   DATA[261,19] := 2.0;
   DATA[261,20] := 148.808;
   DATA[261,21] := 155.9087;
   DATA[261,22] := 1.718643;
   DATA[261,23] := 962.9838;
   DATA[261,24] := 2.0;
   DATA[261,25] := 2.0;
   DATA[261,26] := 7.876058;
   DATA[261,27] := 144.9885;
   DATA[261,28] := 264.0989;
   DATA[261,29] := 12.15073;
   DATA[261,30] := 1.730069;
   DATA[261,31] := 1.257846;
   DATA[261,32] := 0.7351407;
   DATA[261,33] := 0.3077859;
   DATA[261,34] := 2.0;
   DATA[261,35] := 251.0414;
   DATA[261,36] := 1.649953;
   DATA[261,37] := 189.8231;
   DATA[261,38] := 0.000128152;
   DATA[261,39] := 1.0;
   DATA[262,0] := 2.540755;
   DATA[262,1] := 527.243;
   DATA[262,2] := 2.0;
   DATA[262,3] := 2.0;
   DATA[262,4] := 262.0802;
   DATA[262,5] := 8.393873;
   DATA[262,6] := 328.2748;
   DATA[262,7] := 2.444623;
   DATA[262,8] := 2.0;
   DATA[262,9] := 2.0;
   DATA[262,10] := 2.0;
   DATA[262,11] := 19.62033;
   DATA[262,12] := 2.213496;
   DATA[262,13] := 968.2213;
   DATA[262,14] := 1.0;
   DATA[262,15] := 2.0;
   DATA[262,16] := 1.0;
   DATA[262,17] := 1.0;
   DATA[262,18] := 1.0;
   DATA[262,19] := 2.0;
   DATA[262,20] := 148.808;
   DATA[262,21] := 155.9344;
   DATA[262,22] := 1.719284;
   DATA[262,23] := 963.253;
   DATA[262,24] := 2.0;
   DATA[262,25] := 2.0;
   DATA[262,26] := 7.876058;
   DATA[262,27] := 144.9885;
   DATA[262,28] := 264.0989;
   DATA[262,29] := 12.15073;
   DATA[262,30] := 1.73071;
   DATA[262,31] := 1.254515;
   DATA[262,32] := 0.7351407;
   DATA[262,33] := 0.3077859;
   DATA[262,34] := 2.0;
   DATA[262,35] := 251.0414;
   DATA[262,36] := 1.649953;
   DATA[262,37] := 189.8231;
   DATA[262,38] := 0.000128152;
   DATA[262,39] := 1.0;
   DATA[263,0] := 2.577587;
   DATA[263,1] := 527.4393;
   DATA[263,2] := 2.0;
   DATA[263,3] := 2.0;
   DATA[263,4] := 262.0802;
   DATA[263,5] := 8.393873;
   DATA[263,6] := 328.121;
   DATA[263,7] := 2.444623;
   DATA[263,8] := 2.0;
   DATA[263,9] := 2.0;
   DATA[263,10] := 2.0;
   DATA[263,11] := 19.62033;
   DATA[263,12] := 2.214137;
   DATA[263,13] := 968.6218;
   DATA[263,14] := 1.0;
   DATA[263,15] := 2.0;
   DATA[263,16] := 1.0;
   DATA[263,17] := 1.0;
   DATA[263,18] := 1.0;
   DATA[263,19] := 2.0;
   DATA[263,20] := 148.808;
   DATA[263,21] := 155.9344;
   DATA[263,22] := 1.719284;
   DATA[263,23] := 963.4453;
   DATA[263,24] := 2.0;
   DATA[263,25] := 2.0;
   DATA[263,26] := 7.876058;
   DATA[263,27] := 144.9885;
   DATA[263,28] := 264.0989;
   DATA[263,29] := 12.15073;
   DATA[263,30] := 1.73071;
   DATA[263,31] := 1.257205;
   DATA[263,32] := 0.7351407;
   DATA[263,33] := 0.3068251;
   DATA[263,34] := 2.0;
   DATA[263,35] := 251.0414;
   DATA[263,36] := 1.649953;
   DATA[263,37] := 189.8231;
   DATA[263,38] := 0.000128152;
   DATA[263,39] := 1.0;
   DATA[264,0] := 2.6157;
   DATA[264,1] := 527.7534;
   DATA[264,2] := 2.0;
   DATA[264,3] := 2.0;
   DATA[264,4] := 262.0802;
   DATA[264,5] := 8.393873;
   DATA[264,6] := 328.121;
   DATA[264,7] := 2.44411;
   DATA[264,8] := 2.0;
   DATA[264,9] := 2.0;
   DATA[264,10] := 2.0;
   DATA[264,11] := 19.64594;
   DATA[264,12] := 2.214137;
   DATA[264,13] := 968.5818;
   DATA[264,14] := 1.0;
   DATA[264,15] := 2.0;
   DATA[264,16] := 1.0;
   DATA[264,17] := 1.0;
   DATA[264,18] := 1.0;
   DATA[264,19] := 2.0;
   DATA[264,20] := 148.808;
   DATA[264,21] := 155.9344;
   DATA[264,22] := 1.719284;
   DATA[264,23] := 963.4068;
   DATA[264,24] := 2.0;
   DATA[264,25] := 2.0;
   DATA[264,26] := 7.876058;
   DATA[264,27] := 144.9885;
   DATA[264,28] := 264.0989;
   DATA[264,29] := 12.15073;
   DATA[264,30] := 1.729557;
   DATA[264,31] := 1.261944;
   DATA[264,32] := 0.7351407;
   DATA[264,33] := 0.3068251;
   DATA[264,34] := 2.0;
   DATA[264,35] := 251.1055;
   DATA[264,36] := 1.649953;
   DATA[264,37] := 189.8231;
   DATA[264,38] := 0.000128152;
   DATA[264,39] := 1.0;
   DATA[265,0] := 2.637799;
   DATA[265,1] := 527.9496;
   DATA[265,2] := 2.0;
   DATA[265,3] := 2.0;
   DATA[265,4] := 262.0802;
   DATA[265,5] := 8.393873;
   DATA[265,6] := 328.121;
   DATA[265,7] := 2.4427;
   DATA[265,8] := 2.0;
   DATA[265,9] := 2.0;
   DATA[265,10] := 2.0;
   DATA[265,11] := 19.66835;
   DATA[265,12] := 2.214137;
   DATA[265,13] := 968.6218;
   DATA[265,14] := 1.0;
   DATA[265,15] := 2.0;
   DATA[265,16] := 1.0;
   DATA[265,17] := 1.0;
   DATA[265,18] := 1.0;
   DATA[265,19] := 2.0;
   DATA[265,20] := 148.808;
   DATA[265,21] := 155.9344;
   DATA[265,22] := 1.719284;
   DATA[265,23] := 963.1761;
   DATA[265,24] := 2.0;
   DATA[265,25] := 2.0;
   DATA[265,26] := 7.876058;
   DATA[265,27] := 144.9885;
   DATA[265,28] := 264.0989;
   DATA[265,29] := 12.15073;
   DATA[265,30] := 1.729172;
   DATA[265,31] := 1.277699;
   DATA[265,32] := 0.7351407;
   DATA[265,33] := 0.3063127;
   DATA[265,34] := 2.0;
   DATA[265,35] := 251.1055;
   DATA[265,36] := 1.649953;
   DATA[265,37] := 189.8071;
   DATA[265,38] := 0.000128152;
   DATA[265,39] := 1.0;
   DATA[266,0] := 2.656055;
   DATA[266,1] := 527.7534;
   DATA[266,2] := 2.0;
   DATA[266,3] := 2.0;
   DATA[266,4] := 262.0802;
   DATA[266,5] := 8.393873;
   DATA[266,6] := 328.121;
   DATA[266,7] := 2.442316;
   DATA[266,8] := 2.0;
   DATA[266,9] := 2.0;
   DATA[266,10] := 2.0;
   DATA[266,11] := 19.66835;
   DATA[266,12] := 2.214137;
   DATA[266,13] := 968.742;
   DATA[266,14] := 1.0;
   DATA[266,15] := 2.0;
   DATA[266,16] := 1.0;
   DATA[266,17] := 1.0;
   DATA[266,18] := 1.0;
   DATA[266,19] := 2.0;
   DATA[266,20] := 148.808;
   DATA[266,21] := 155.9344;
   DATA[266,22] := 1.71813;
   DATA[266,23] := 963.2145;
   DATA[266,24] := 2.0;
   DATA[266,25] := 2.0;
   DATA[266,26] := 7.876058;
   DATA[266,27] := 144.9885;
   DATA[266,28] := 264.0989;
   DATA[266,29] := 12.15073;
   DATA[266,30] := 1.729172;
   DATA[266,31] := 1.281286;
   DATA[266,32] := 0.7351407;
   DATA[266,33] := 0.3063127;
   DATA[266,34] := 2.0;
   DATA[266,35] := 251.1055;
   DATA[266,36] := 1.649953;
   DATA[266,37] := 189.8071;
   DATA[266,38] := 0.000128152;
   DATA[266,39] := 1.0;
   DATA[267,0] := 2.658617;
   DATA[267,1] := 527.4393;
   DATA[267,2] := 2.0;
   DATA[267,3] := 2.0;
   DATA[267,4] := 262.0802;
   DATA[267,5] := 8.393873;
   DATA[267,6] := 328.121;
   DATA[267,7] := 2.442316;
   DATA[267,8] := 2.0;
   DATA[267,9] := 2.0;
   DATA[267,10] := 2.0;
   DATA[267,11] := 19.66835;
   DATA[267,12] := 2.214137;
   DATA[267,13] := 968.8221;
   DATA[267,14] := 1.0;
   DATA[267,15] := 2.0;
   DATA[267,16] := 1.0;
   DATA[267,17] := 1.0;
   DATA[267,18] := 1.0;
   DATA[267,19] := 2.0;
   DATA[267,20] := 148.808;
   DATA[267,21] := 155.9344;
   DATA[267,22] := 1.71813;
   DATA[267,23] := 963.1761;
   DATA[267,24] := 2.0;
   DATA[267,25] := 2.0;
   DATA[267,26] := 7.876058;
   DATA[267,27] := 144.9885;
   DATA[267,28] := 264.0028;
   DATA[267,29] := 12.15073;
   DATA[267,30] := 1.729172;
   DATA[267,31] := 1.290637;
   DATA[267,32] := 0.7351407;
   DATA[267,33] := 0.3063127;
   DATA[267,34] := 2.0;
   DATA[267,35] := 251.1055;
   DATA[267,36] := 1.649953;
   DATA[267,37] := 189.8071;
   DATA[267,38] := 0.000128152;
   DATA[267,39] := 1.0;
   DATA[268,0] := 2.638119;
   DATA[268,1] := 527.4393;
   DATA[268,2] := 2.0;
   DATA[268,3] := 2.0;
   DATA[268,4] := 262.0802;
   DATA[268,5] := 8.393873;
   DATA[268,6] := 328.121;
   DATA[268,7] := 2.442316;
   DATA[268,8] := 2.0;
   DATA[268,9] := 2.0;
   DATA[268,10] := 2.0;
   DATA[268,11] := 19.70677;
   DATA[268,12] := 2.212856;
   DATA[268,13] := 968.9824;
   DATA[268,14] := 1.0;
   DATA[268,15] := 2.0;
   DATA[268,16] := 1.0;
   DATA[268,17] := 1.0;
   DATA[268,18] := 1.0;
   DATA[268,19] := 2.0;
   DATA[268,20] := 148.808;
   DATA[268,21] := 155.9344;
   DATA[268,22] := 1.71813;
   DATA[268,23] := 963.2914;
   DATA[268,24] := 2.0;
   DATA[268,25] := 2.0;
   DATA[268,26] := 7.876058;
   DATA[268,27] := 144.9885;
   DATA[268,28] := 263.8105;
   DATA[268,29] := 12.15073;
   DATA[268,30] := 1.729172;
   DATA[268,31] := 1.301524;
   DATA[268,32] := 0.7351407;
   DATA[268,33] := 0.3063127;
   DATA[268,34] := 2.0;
   DATA[268,35] := 251.1055;
   DATA[268,36] := 1.649953;
   DATA[268,37] := 189.8071;
   DATA[268,38] := 0.000128152;
   DATA[268,39] := 1.0;
   DATA[269,0] := 2.624027;
   DATA[269,1] := 527.6748;
   DATA[269,2] := 2.0;
   DATA[269,3] := 2.0;
   DATA[269,4] := 262.0802;
   DATA[269,5] := 8.393873;
   DATA[269,6] := 328.121;
   DATA[269,7] := 2.442316;
   DATA[269,8] := 2.0;
   DATA[269,9] := 2.0;
   DATA[269,10] := 2.0;
   DATA[269,11] := 19.74198;
   DATA[269,12] := 2.2126;
   DATA[269,13] := 968.8221;
   DATA[269,14] := 1.0;
   DATA[269,15] := 2.0;
   DATA[269,16] := 1.0;
   DATA[269,17] := 1.0;
   DATA[269,18] := 1.0;
   DATA[269,19] := 2.0;
   DATA[269,20] := 148.808;
   DATA[269,21] := 155.9344;
   DATA[269,22] := 1.717489;
   DATA[269,23] := 963.4837;
   DATA[269,24] := 2.0;
   DATA[269,25] := 2.0;
   DATA[269,26] := 7.876058;
   DATA[269,27] := 144.9885;
   DATA[269,28] := 263.8105;
   DATA[269,29] := 12.15073;
   DATA[269,30] := 1.726737;
   DATA[269,31] := 1.301524;
   DATA[269,32] := 0.7351407;
   DATA[269,33] := 0.3072094;
   DATA[269,34] := 2.0;
   DATA[269,35] := 251.1055;
   DATA[269,36] := 1.649953;
   DATA[269,37] := 189.727;
   DATA[269,38] := 0.000128152;
   DATA[269,39] := 1.0;
   DATA[270,0] := 2.620184;
   DATA[270,1] := 527.5963;
   DATA[270,2] := 2.0;
   DATA[270,3] := 2.0;
   DATA[270,4] := 262.0802;
   DATA[270,5] := 8.393873;
   DATA[270,6] := 328.121;
   DATA[270,7] := 2.441803;
   DATA[270,8] := 2.0;
   DATA[270,9] := 2.0;
   DATA[270,10] := 2.0;
   DATA[270,11] := 19.77399;
   DATA[270,12] := 2.2126;
   DATA[270,13] := 968.8622;
   DATA[270,14] := 1.0;
   DATA[270,15] := 2.0;
   DATA[270,16] := 1.0;
   DATA[270,17] := 1.0;
   DATA[270,18] := 1.0;
   DATA[270,19] := 2.0;
   DATA[270,20] := 148.808;
   DATA[270,21] := 155.9344;
   DATA[270,22] := 1.715824;
   DATA[270,23] := 963.7529;
   DATA[270,24] := 2.0;
   DATA[270,25] := 2.0;
   DATA[270,26] := 7.876058;
   DATA[270,27] := 144.9885;
   DATA[270,28] := 263.8105;
   DATA[270,29] := 12.15073;
   DATA[270,30] := 1.726737;
   DATA[270,31] := 1.312284;
   DATA[270,32] := 0.7351407;
   DATA[270,33] := 0.3072735;
   DATA[270,34] := 2.0;
   DATA[270,35] := 251.1055;
   DATA[270,36] := 1.649953;
   DATA[270,37] := 189.6789;
   DATA[270,38] := 0.000128152;
   DATA[270,39] := 1.0;
   DATA[271,0] := 2.609935;
   DATA[271,1] := 527.9496;
   DATA[271,2] := 2.0;
   DATA[271,3] := 2.0;
   DATA[271,4] := 262.0802;
   DATA[271,5] := 8.393873;
   DATA[271,6] := 328.121;
   DATA[271,7] := 2.439625;
   DATA[271,8] := 2.0;
   DATA[271,9] := 2.0;
   DATA[271,10] := 2.0;
   DATA[271,11] := 19.77399;
   DATA[271,12] := 2.211447;
   DATA[271,13] := 969.5831;
   DATA[271,14] := 1.0;
   DATA[271,15] := 2.0;
   DATA[271,16] := 1.0;
   DATA[271,17] := 1.0;
   DATA[271,18] := 1.0;
   DATA[271,19] := 2.0;
   DATA[271,20] := 148.808;
   DATA[271,21] := 155.9344;
   DATA[271,22] := 1.715824;
   DATA[271,23] := 963.676;
   DATA[271,24] := 2.0;
   DATA[271,25] := 2.0;
   DATA[271,26] := 7.876058;
   DATA[271,27] := 144.8603;
   DATA[271,28] := 263.8105;
   DATA[271,29] := 12.15073;
   DATA[271,30] := 1.728788;
   DATA[271,31] := 1.30716;
   DATA[271,32] := 0.7351407;
   DATA[271,33] := 0.3072735;
   DATA[271,34] := 2.0;
   DATA[271,35] := 250.9613;
   DATA[271,36] := 1.649953;
   DATA[271,37] := 189.6629;
   DATA[271,38] := 0.000128152;
   DATA[271,39] := 1.0;
   DATA[272,0] := 2.598085;
   DATA[272,1] := 527.8711;
   DATA[272,2] := 2.0;
   DATA[272,3] := 2.0;
   DATA[272,4] := 262.0802;
   DATA[272,5] := 8.393873;
   DATA[272,6] := 328.3517;
   DATA[272,7] := 2.439625;
   DATA[272,8] := 2.0;
   DATA[272,9] := 2.0;
   DATA[272,10] := 2.0;
   DATA[272,11] := 19.76439;
   DATA[272,12] := 2.209653;
   DATA[272,13] := 969.463;
   DATA[272,14] := 1.0;
   DATA[272,15] := 2.0;
   DATA[272,16] := 1.0;
   DATA[272,17] := 1.0;
   DATA[272,18] := 1.0;
   DATA[272,19] := 2.0;
   DATA[272,20] := 148.808;
   DATA[272,21] := 155.9344;
   DATA[272,22] := 1.715824;
   DATA[272,23] := 963.9451;
   DATA[272,24] := 2.0;
   DATA[272,25] := 2.0;
   DATA[272,26] := 7.876058;
   DATA[272,27] := 144.8603;
   DATA[272,28] := 263.8105;
   DATA[272,29] := 12.15073;
   DATA[272,30] := 1.728788;
   DATA[272,31] := 1.288075;
   DATA[272,32] := 0.7351407;
   DATA[272,33] := 0.306761;
   DATA[272,34] := 2.0;
   DATA[272,35] := 250.8972;
   DATA[272,36] := 1.649953;
   DATA[272,37] := 189.6629;
   DATA[272,38] := 0.000128152;
   DATA[272,39] := 1.0;
   DATA[273,0] := 2.572783;
   DATA[273,1] := 527.7926;
   DATA[273,2] := 2.0;
   DATA[273,3] := 2.0;
   DATA[273,4] := 262.0802;
   DATA[273,5] := 8.392271;
   DATA[273,6] := 328.3773;
   DATA[273,7] := 2.441803;
   DATA[273,8] := 2.0;
   DATA[273,9] := 2.0;
   DATA[273,10] := 2.0;
   DATA[273,11] := 19.76439;
   DATA[273,12] := 2.208884;
   DATA[273,13] := 969.3829;
   DATA[273,14] := 1.0;
   DATA[273,15] := 2.0;
   DATA[273,16] := 1.0;
   DATA[273,17] := 1.0;
   DATA[273,18] := 1.0;
   DATA[273,19] := 2.0;
   DATA[273,20] := 148.808;
   DATA[273,21] := 155.9344;
   DATA[273,22] := 1.717105;
   DATA[273,23] := 963.8298;
   DATA[273,24] := 2.0;
   DATA[273,25] := 2.0;
   DATA[273,26] := 7.876058;
   DATA[273,27] := 144.8603;
   DATA[273,28] := 263.8105;
   DATA[273,29] := 12.15073;
   DATA[273,30] := 1.728788;
   DATA[273,31] := 1.281927;
   DATA[273,32] := 0.7351407;
   DATA[273,33] := 0.306761;
   DATA[273,34] := 2.0;
   DATA[273,35] := 250.8972;
   DATA[273,36] := 1.649953;
   DATA[273,37] := 189.6629;
   DATA[273,38] := 0.000128152;
   DATA[273,39] := 1.0;
   DATA[274,0] := 2.561573;
   DATA[274,1] := 527.8711;
   DATA[274,2] := 2.0;
   DATA[274,3] := 2.0;
   DATA[274,4] := 262.0802;
   DATA[274,5] := 8.392271;
   DATA[274,6] := 328.3773;
   DATA[274,7] := 2.442444;
   DATA[274,8] := 2.0;
   DATA[274,9] := 2.0;
   DATA[274,10] := 2.0;
   DATA[274,11] := 19.73238;
   DATA[274,12] := 2.208884;
   DATA[274,13] := 969.3428;
   DATA[274,14] := 1.0;
   DATA[274,15] := 2.0;
   DATA[274,16] := 1.0;
   DATA[274,17] := 1.0;
   DATA[274,18] := 1.0;
   DATA[274,19] := 2.0;
   DATA[274,20] := 148.808;
   DATA[274,21] := 155.9344;
   DATA[274,22] := 1.717489;
   DATA[274,23] := 964.3297;
   DATA[274,24] := 2.0;
   DATA[274,25] := 2.0;
   DATA[274,26] := 7.876058;
   DATA[274,27] := 144.8603;
   DATA[274,28] := 264.0989;
   DATA[274,29] := 12.15073;
   DATA[274,30] := 1.728788;
   DATA[274,31] := 1.271935;
   DATA[274,32] := 0.7351407;
   DATA[274,33] := 0.3072094;
   DATA[274,34] := 2.0;
   DATA[274,35] := 250.8972;
   DATA[274,36] := 1.649953;
   DATA[274,37] := 189.6629;
   DATA[274,38] := 0.000128152;
   DATA[274,39] := 1.0;
   DATA[275,0] := 2.541716;
   DATA[275,1] := 528.0281;
   DATA[275,2] := 2.0;
   DATA[275,3] := 2.0;
   DATA[275,4] := 262.0802;
   DATA[275,5] := 8.39131;
   DATA[275,6] := 328.3773;
   DATA[275,7] := 2.442444;
   DATA[275,8] := 2.0;
   DATA[275,9] := 2.0;
   DATA[275,10] := 2.0;
   DATA[275,11] := 19.73238;
   DATA[275,12] := 2.208884;
   DATA[275,13] := 969.5431;
   DATA[275,14] := 1.0;
   DATA[275,15] := 2.0;
   DATA[275,16] := 1.0;
   DATA[275,17] := 1.0;
   DATA[275,18] := 1.0;
   DATA[275,19] := 2.0;
   DATA[275,20] := 148.808;
   DATA[275,21] := 155.9344;
   DATA[275,22] := 1.717489;
   DATA[275,23] := 964.3681;
   DATA[275,24] := 2.0;
   DATA[275,25] := 2.0;
   DATA[275,26] := 7.876058;
   DATA[275,27] := 144.8603;
   DATA[275,28] := 264.0989;
   DATA[275,29] := 12.11228;
   DATA[275,30] := 1.728788;
   DATA[275,31] := 1.275906;
   DATA[275,32] := 0.7351407;
   DATA[275,33] := 0.3074016;
   DATA[275,34] := 2.0;
   DATA[275,35] := 250.8972;
   DATA[275,36] := 1.649953;
   DATA[275,37] := 189.6629;
   DATA[275,38] := 0.000128152;
   DATA[275,39] := 1.0;
   DATA[276,0] := 2.528264;
   DATA[276,1] := 528.5776;
   DATA[276,2] := 2.0;
   DATA[276,3] := 2.0;
   DATA[276,4] := 262.0802;
   DATA[276,5] := 8.39131;
   DATA[276,6] := 328.2492;
   DATA[276,7] := 2.441547;
   DATA[276,8] := 2.0;
   DATA[276,9] := 2.0;
   DATA[276,10] := 2.0;
   DATA[276,11] := 19.73238;
   DATA[276,12] := 2.208884;
   DATA[276,13] := 969.463;
   DATA[276,14] := 1.0;
   DATA[276,15] := 2.0;
   DATA[276,16] := 1.0;
   DATA[276,17] := 1.0;
   DATA[276,18] := 1.0;
   DATA[276,19] := 2.0;
   DATA[276,20] := 148.808;
   DATA[276,21] := 155.9344;
   DATA[276,22] := 1.717489;
   DATA[276,23] := 964.4066;
   DATA[276,24] := 2.0;
   DATA[276,25] := 2.0;
   DATA[276,26] := 7.876058;
   DATA[276,27] := 144.8603;
   DATA[276,28] := 264.0989;
   DATA[276,29] := 12.11228;
   DATA[276,30] := 1.728788;
   DATA[276,31] := 1.291277;
   DATA[276,32] := 0.7351407;
   DATA[276,33] := 0.3074016;
   DATA[276,34] := 2.0;
   DATA[276,35] := 250.8972;
   DATA[276,36] := 1.649953;
   DATA[276,37] := 189.6629;
   DATA[276,38] := 0.000128152;
   DATA[276,39] := 1.0;
   DATA[277,0] := 2.505204;
   DATA[277,1] := 529.0486;
   DATA[277,2] := 2.0;
   DATA[277,3] := 2.0;
   DATA[277,4] := 262.0802;
   DATA[277,5] := 8.39131;
   DATA[277,6] := 328.2492;
   DATA[277,7] := 2.439881;
   DATA[277,8] := 2.0;
   DATA[277,9] := 2.0;
   DATA[277,10] := 2.0;
   DATA[277,11] := 19.73238;
   DATA[277,12] := 2.210934;
   DATA[277,13] := 969.1826;
   DATA[277,14] := 1.0;
   DATA[277,15] := 2.0;
   DATA[277,16] := 1.0;
   DATA[277,17] := 1.0;
   DATA[277,18] := 1.0;
   DATA[277,19] := 2.0;
   DATA[277,20] := 148.808;
   DATA[277,21] := 155.9344;
   DATA[277,22] := 1.717489;
   DATA[277,23] := 964.5988;
   DATA[277,24] := 2.0;
   DATA[277,25] := 2.0;
   DATA[277,26] := 7.876058;
   DATA[277,27] := 144.8603;
   DATA[277,28] := 264.0669;
   DATA[277,29] := 12.11228;
   DATA[277,30] := 1.728916;
   DATA[277,31] := 1.287434;
   DATA[277,32] := 0.7351407;
   DATA[277,33] := 0.3068891;
   DATA[277,34] := 2.0;
   DATA[277,35] := 250.8972;
   DATA[277,36] := 1.649953;
   DATA[277,37] := 189.6629;
   DATA[277,38] := 0.000128152;
   DATA[277,39] := 1.0;
   DATA[278,0] := 2.491432;
   DATA[278,1] := 528.7739;
   DATA[278,2] := 2.0;
   DATA[278,3] := 2.0;
   DATA[278,4] := 262.0802;
   DATA[278,5] := 8.39131;
   DATA[278,6] := 328.2492;
   DATA[278,7] := 2.439881;
   DATA[278,8] := 2.0;
   DATA[278,9] := 2.0;
   DATA[278,10] := 2.0;
   DATA[278,11] := 19.73238;
   DATA[278,12] := 2.2126;
   DATA[278,13] := 969.463;
   DATA[278,14] := 1.0;
   DATA[278,15] := 2.0;
   DATA[278,16] := 1.0;
   DATA[278,17] := 1.0;
   DATA[278,18] := 1.0;
   DATA[278,19] := 2.0;
   DATA[278,20] := 148.808;
   DATA[278,21] := 155.9344;
   DATA[278,22] := 1.717489;
   DATA[278,23] := 964.8295;
   DATA[278,24] := 2.0;
   DATA[278,25] := 2.0;
   DATA[278,26] := 7.876058;
   DATA[278,27] := 144.8603;
   DATA[278,28] := 263.9067;
   DATA[278,29] := 12.11228;
   DATA[278,30] := 1.729557;
   DATA[278,31] := 1.28167;
   DATA[278,32] := 0.7351407;
   DATA[278,33] := 0.3065048;
   DATA[278,34] := 2.0;
   DATA[278,35] := 250.8972;
   DATA[278,36] := 1.649953;
   DATA[278,37] := 189.6629;
   DATA[278,38] := 0.000128152;
   DATA[278,39] := 1.0;
   DATA[279,0] := 2.471575;
   DATA[279,1] := 528.4599;
   DATA[279,2] := 2.0;
   DATA[279,3] := 2.0;
   DATA[279,4] := 262.0802;
   DATA[279,5] := 8.39131;
   DATA[279,6] := 328.2492;
   DATA[279,7] := 2.439881;
   DATA[279,8] := 2.0;
   DATA[279,9] := 2.0;
   DATA[279,10] := 2.0;
   DATA[279,11] := 19.73238;
   DATA[279,12] := 2.212984;
   DATA[279,13] := 969.5831;
   DATA[279,14] := 1.0;
   DATA[279,15] := 2.0;
   DATA[279,16] := 1.0;
   DATA[279,17] := 1.0;
   DATA[279,18] := 1.0;
   DATA[279,19] := 2.0;
   DATA[279,20] := 148.808;
   DATA[279,21] := 155.9344;
   DATA[279,22] := 1.717489;
   DATA[279,23] := 965.1371;
   DATA[279,24] := 2.0;
   DATA[279,25] := 2.0;
   DATA[279,26] := 7.876058;
   DATA[279,27] := 144.8603;
   DATA[279,28] := 263.9067;
   DATA[279,29] := 12.11228;
   DATA[279,30] := 1.729557;
   DATA[279,31] := 1.287306;
   DATA[279,32] := 0.7351407;
   DATA[279,33] := 0.3065048;
   DATA[279,34] := 2.0;
   DATA[279,35] := 250.8972;
   DATA[279,36] := 1.649953;
   DATA[279,37] := 189.6629;
   DATA[279,38] := 0.000128152;
   DATA[279,39] := 1.0;
   DATA[280,0] := 2.471575;
   DATA[280,1] := 528.4599;
   DATA[280,2] := 2.0;
   DATA[280,3] := 2.0;
   DATA[280,4] := 262.0802;
   DATA[280,5] := 8.39131;
   DATA[280,6] := 328.2492;
   DATA[280,7] := 2.439881;
   DATA[280,8] := 2.0;
   DATA[280,9] := 2.0;
   DATA[280,10] := 2.0;
   DATA[280,11] := 19.73238;
   DATA[280,12] := 2.212984;
   DATA[280,13] := 969.5831;
   DATA[280,14] := 1.0;
   DATA[280,15] := 2.0;
   DATA[280,16] := 1.0;
   DATA[280,17] := 1.0;
   DATA[280,18] := 1.0;
   DATA[280,19] := 2.0;
   DATA[280,20] := 148.808;
   DATA[280,21] := 155.9344;
   DATA[280,22] := 1.717489;
   DATA[280,23] := 965.1371;
   DATA[280,24] := 2.0;
   DATA[280,25] := 2.0;
   DATA[280,26] := 7.876058;
   DATA[280,27] := 144.8603;
   DATA[280,28] := 263.9067;
   DATA[280,29] := 12.11228;
   DATA[280,30] := 1.729557;
   DATA[280,31] := 1.287306;
   DATA[280,32] := 0.7351407;
   DATA[280,33] := 0.3065048;
   DATA[280,34] := 2.0;
   DATA[280,35] := 250.8972;
   DATA[280,36] := 1.649953;
   DATA[280,37] := 189.6629;
   DATA[280,38] := 0.000128152;
   DATA[280,39] := 1.0;
   DATA[281,0] := 2.460366;
   DATA[281,1] := 528.5384;
   DATA[281,2] := 2.0;
   DATA[281,3] := 2.0;
   DATA[281,4] := 262.0802;
   DATA[281,5] := 8.39131;
   DATA[281,6] := 328.2492;
   DATA[281,7] := 2.439881;
   DATA[281,8] := 2.0;
   DATA[281,9] := 2.0;
   DATA[281,10] := 2.0;
   DATA[281,11] := 19.73558;
   DATA[281,12] := 2.212984;
   DATA[281,13] := 969.5431;
   DATA[281,14] := 1.0;
   DATA[281,15] := 2.0;
   DATA[281,16] := 1.0;
   DATA[281,17] := 1.0;
   DATA[281,18] := 1.0;
   DATA[281,19] := 2.0;
   DATA[281,20] := 148.808;
   DATA[281,21] := 155.9344;
   DATA[281,22] := 1.717489;
   DATA[281,23] := 965.4063;
   DATA[281,24] := 2.0;
   DATA[281,25] := 2.0;
   DATA[281,26] := 7.876058;
   DATA[281,27] := 144.8603;
   DATA[281,28] := 263.9067;
   DATA[281,29] := 12.11228;
   DATA[281,30] := 1.729557;
   DATA[281,31] := 1.292046;
   DATA[281,32] := 0.7351407;
   DATA[281,33] := 0.3065048;
   DATA[281,34] := 2.0;
   DATA[281,35] := 250.8972;
   DATA[281,36] := 1.649953;
   DATA[281,37] := 189.6629;
   DATA[281,38] := 0.000128152;
   DATA[281,39] := 1.0;
   DATA[282,0] := 2.447555;
   DATA[282,1] := 528.3421;
   DATA[282,2] := 2.0;
   DATA[282,3] := 2.0;
   DATA[282,4] := 262.0802;
   DATA[282,5] := 8.39131;
   DATA[282,6] := 328.2492;
   DATA[282,7] := 2.439881;
   DATA[282,8] := 2.0;
   DATA[282,9] := 2.0;
   DATA[282,10] := 2.0;
   DATA[282,11] := 19.82841;
   DATA[282,12] := 2.212984;
   DATA[282,13] := 969.463;
   DATA[282,14] := 1.0;
   DATA[282,15] := 2.0;
   DATA[282,16] := 1.0;
   DATA[282,17] := 1.0;
   DATA[282,18] := 1.0;
   DATA[282,19] := 2.0;
   DATA[282,20] := 148.808;
   DATA[282,21] := 156.0625;
   DATA[282,22] := 1.717489;
   DATA[282,23] := 965.7139;
   DATA[282,24] := 2.0;
   DATA[282,25] := 2.0;
   DATA[282,26] := 7.876058;
   DATA[282,27] := 144.8603;
   DATA[282,28] := 263.9067;
   DATA[282,29] := 12.11228;
   DATA[282,30] := 1.729557;
   DATA[282,31] := 1.309082;
   DATA[282,32] := 0.7351407;
   DATA[282,33] := 0.3065048;
   DATA[282,34] := 2.0;
   DATA[282,35] := 250.8972;
   DATA[282,36] := 1.649953;
   DATA[282,37] := 189.6629;
   DATA[282,38] := 0.000128152;
   DATA[282,39] := 1.0;
   DATA[283,0] := 2.434423;
   DATA[283,1] := 528.1459;
   DATA[283,2] := 2.0;
   DATA[283,3] := 2.0;
   DATA[283,4] := 262.0802;
   DATA[283,5] := 8.39131;
   DATA[283,6] := 328.2492;
   DATA[283,7] := 2.439881;
   DATA[283,8] := 2.0;
   DATA[283,9] := 2.0;
   DATA[283,10] := 2.0;
   DATA[283,11] := 19.84762;
   DATA[283,12] := 2.210166;
   DATA[283,13] := 969.8635;
   DATA[283,14] := 1.0;
   DATA[283,15] := 2.0;
   DATA[283,16] := 1.0;
   DATA[283,17] := 1.0;
   DATA[283,18] := 1.0;
   DATA[283,19] := 2.0;
   DATA[283,20] := 148.808;
   DATA[283,21] := 156.0625;
   DATA[283,22] := 1.717489;
   DATA[283,23] := 965.7139;
   DATA[283,24] := 2.0;
   DATA[283,25] := 2.0;
   DATA[283,26] := 7.876058;
   DATA[283,27] := 144.8603;
   DATA[283,28] := 263.9067;
   DATA[283,29] := 12.11228;
   DATA[283,30] := 1.72725;
   DATA[283,31] := 1.321634;
   DATA[283,32] := 0.7351407;
   DATA[283,33] := 0.3065048;
   DATA[283,34] := 2.0;
   DATA[283,35] := 250.9453;
   DATA[283,36] := 1.649953;
   DATA[283,37] := 189.759;
   DATA[283,38] := 0.000128152;
   DATA[283,39] := 1.0;
   DATA[284,0] := 2.428338;
   DATA[284,1] := 528.0674;
   DATA[284,2] := 2.0;
   DATA[284,3] := 2.0;
   DATA[284,4] := 262.0802;
   DATA[284,5] := 8.39131;
   DATA[284,6] := 328.2492;
   DATA[284,7] := 2.439881;
   DATA[284,8] := 2.0;
   DATA[284,9] := 2.0;
   DATA[284,10] := 2.0;
   DATA[284,11] := 19.7868;
   DATA[284,12] := 2.209525;
   DATA[284,13] := 969.6633;
   DATA[284,14] := 1.0;
   DATA[284,15] := 2.0;
   DATA[284,16] := 1.0;
   DATA[284,17] := 1.0;
   DATA[284,18] := 1.0;
   DATA[284,19] := 2.0;
   DATA[284,20] := 148.808;
   DATA[284,21] := 156.0625;
   DATA[284,22] := 1.717489;
   DATA[284,23] := 965.7524;
   DATA[284,24] := 2.0;
   DATA[284,25] := 2.0;
   DATA[284,26] := 7.876058;
   DATA[284,27] := 144.8603;
   DATA[284,28] := 263.9067;
   DATA[284,29] := 12.11228;
   DATA[284,30] := 1.72725;
   DATA[284,31] := 1.317536;
   DATA[284,32] := 0.7351407;
   DATA[284,33] := 0.3065048;
   DATA[284,34] := 2.0;
   DATA[284,35] := 251.0574;
   DATA[284,36] := 1.649953;
   DATA[284,37] := 189.759;
   DATA[284,38] := 0.000128152;
   DATA[284,39] := 1.0;
   DATA[285,0] := 2.428338;
   DATA[285,1] := 528.2244;
   DATA[285,2] := 2.0;
   DATA[285,3] := 2.0;
   DATA[285,4] := 262.0802;
   DATA[285,5] := 8.39131;
   DATA[285,6] := 328.2492;
   DATA[285,7] := 2.439881;
   DATA[285,8] := 2.0;
   DATA[285,9] := 2.0;
   DATA[285,10] := 2.0;
   DATA[285,11] := 19.75479;
   DATA[285,12] := 2.209525;
   DATA[285,13] := 970.184;
   DATA[285,14] := 1.0;
   DATA[285,15] := 2.0;
   DATA[285,16] := 1.0;
   DATA[285,17] := 1.0;
   DATA[285,18] := 1.0;
   DATA[285,19] := 2.0;
   DATA[285,20] := 148.808;
   DATA[285,21] := 156.0625;
   DATA[285,22] := 1.717489;
   DATA[285,23] := 965.8677;
   DATA[285,24] := 2.0;
   DATA[285,25] := 2.0;
   DATA[285,26] := 7.876058;
   DATA[285,27] := 144.8603;
   DATA[285,28] := 263.9067;
   DATA[285,29] := 12.11228;
   DATA[285,30] := 1.72725;
   DATA[285,31] := 1.311003;
   DATA[285,32] := 0.7351407;
   DATA[285,33] := 0.3065048;
   DATA[285,34] := 2.0;
   DATA[285,35] := 251.0574;
   DATA[285,36] := 1.649953;
   DATA[285,37] := 189.759;
   DATA[285,38] := 0.000128152;
   DATA[285,39] := 1.0;
   DATA[286,0] := 2.447555;
   DATA[286,1] := 528.0674;
   DATA[286,2] := 2.0;
   DATA[286,3] := 2.0;
   DATA[286,4] := 262.0802;
   DATA[286,5] := 8.39131;
   DATA[286,6] := 328.2492;
   DATA[286,7] := 2.440521;
   DATA[286,8] := 2.0;
   DATA[286,9] := 2.0;
   DATA[286,10] := 2.0;
   DATA[286,11] := 19.75479;
   DATA[286,12] := 2.209525;
   DATA[286,13] := 970.0638;
   DATA[286,14] := 1.0;
   DATA[286,15] := 2.0;
   DATA[286,16] := 1.0;
   DATA[286,17] := 1.0;
   DATA[286,18] := 1.0;
   DATA[286,19] := 2.0;
   DATA[286,20] := 148.808;
   DATA[286,21] := 156.0625;
   DATA[286,22] := 1.719924;
   DATA[286,23] := 965.4832;
   DATA[286,24] := 2.0;
   DATA[286,25] := 2.0;
   DATA[286,26] := 7.876058;
   DATA[286,27] := 144.8603;
   DATA[286,28] := 263.9067;
   DATA[286,29] := 12.11228;
   DATA[286,30] := 1.72725;
   DATA[286,31] := 1.301652;
   DATA[286,32] := 0.7351407;
   DATA[286,33] := 0.3065048;
   DATA[286,34] := 2.0;
   DATA[286,35] := 251.0574;
   DATA[286,36] := 1.649953;
   DATA[286,37] := 189.759;
   DATA[286,38] := 0.000128152;
   DATA[286,39] := 1.0;
   DATA[287,0] := 2.5004;
   DATA[287,1] := 528.6561;
   DATA[287,2] := 2.0;
   DATA[287,3] := 2.0;
   DATA[287,4] := 262.0802;
   DATA[287,5] := 8.39131;
   DATA[287,6] := 328.2492;
   DATA[287,7] := 2.440521;
   DATA[287,8] := 2.0;
   DATA[287,9] := 2.0;
   DATA[287,10] := 2.0;
   DATA[287,11] := 19.75479;
   DATA[287,12] := 2.209525;
   DATA[287,13] := 970.5444;
   DATA[287,14] := 1.0;
   DATA[287,15] := 2.0;
   DATA[287,16] := 1.0;
   DATA[287,17] := 1.0;
   DATA[287,18] := 1.0;
   DATA[287,19] := 2.0;
   DATA[287,20] := 148.808;
   DATA[287,21] := 156.0625;
   DATA[287,22] := 1.720437;
   DATA[287,23] := 965.4832;
   DATA[287,24] := 2.0;
   DATA[287,25] := 2.0;
   DATA[287,26] := 7.876058;
   DATA[287,27] := 144.8603;
   DATA[287,28] := 263.9067;
   DATA[287,29] := 12.11228;
   DATA[287,30] := 1.72725;
   DATA[287,31] := 1.301652;
   DATA[287,32] := 0.7351407;
   DATA[287,33] := 0.3065048;
   DATA[287,34] := 2.0;
   DATA[287,35] := 251.0574;
   DATA[287,36] := 1.649953;
   DATA[287,37] := 189.759;
   DATA[287,38] := 0.000128152;
   DATA[287,39] := 1.0;
   DATA[288,0] := 2.544919;
   DATA[288,1] := 528.6561;
   DATA[288,2] := 2.0;
   DATA[288,3] := 2.0;
   DATA[288,4] := 262.0802;
   DATA[288,5] := 8.39131;
   DATA[288,6] := 328.2492;
   DATA[288,7] := 2.441547;
   DATA[288,8] := 2.0;
   DATA[288,9] := 2.0;
   DATA[288,10] := 2.0;
   DATA[288,11] := 19.71957;
   DATA[288,12] := 2.209525;
   DATA[288,13] := 970.4644;
   DATA[288,14] := 1.0;
   DATA[288,15] := 2.0;
   DATA[288,16] := 1.0;
   DATA[288,17] := 1.0;
   DATA[288,18] := 1.0;
   DATA[288,19] := 2.0;
   DATA[288,20] := 148.808;
   DATA[288,21] := 156.0625;
   DATA[288,22] := 1.720437;
   DATA[288,23] := 965.4832;
   DATA[288,24] := 2.0;
   DATA[288,25] := 2.0;
   DATA[288,26] := 7.876058;
   DATA[288,27] := 144.8603;
   DATA[288,28] := 263.9067;
   DATA[288,29] := 12.11228;
   DATA[288,30] := 1.72725;
   DATA[288,31] := 1.310363;
   DATA[288,32] := 0.7351407;
   DATA[288,33] := 0.3065048;
   DATA[288,34] := 2.0;
   DATA[288,35] := 251.0574;
   DATA[288,36] := 1.649953;
   DATA[288,37] := 189.759;
   DATA[288,38] := 0.000128152;
   DATA[288,39] := 1.0;
   DATA[289,0] := 2.588476;
   DATA[289,1] := 528.9309;
   DATA[289,2] := 2.0;
   DATA[289,3] := 2.0;
   DATA[289,4] := 262.1443;
   DATA[289,5] := 8.39131;
   DATA[289,6] := 328.2492;
   DATA[289,7] := 2.442828;
   DATA[289,8] := 2.0;
   DATA[289,9] := 2.0;
   DATA[289,10] := 2.0;
   DATA[289,11] := 19.68756;
   DATA[289,12] := 2.21119;
   DATA[289,13] := 970.4243;
   DATA[289,14] := 1.0;
   DATA[289,15] := 2.0;
   DATA[289,16] := 1.0;
   DATA[289,17] := 1.0;
   DATA[289,18] := 1.0;
   DATA[289,19] := 2.0;
   DATA[289,20] := 148.808;
   DATA[289,21] := 156.0625;
   DATA[289,22] := 1.720437;
   DATA[289,23] := 965.7139;
   DATA[289,24] := 2.0;
   DATA[289,25] := 2.0;
   DATA[289,26] := 7.876058;
   DATA[289,27] := 144.8603;
   DATA[289,28] := 263.9067;
   DATA[289,29] := 12.11228;
   DATA[289,30] := 1.726865;
   DATA[289,31] := 1.311387;
   DATA[289,32] := 0.7351407;
   DATA[289,33] := 0.3065048;
   DATA[289,34] := 2.0;
   DATA[289,35] := 251.2657;
   DATA[289,36] := 1.649953;
   DATA[289,37] := 189.9193;
   DATA[289,38] := 0.000128152;
   DATA[289,39] := 1.0;
   DATA[290,0] := 2.619223;
   DATA[290,1] := 529.0486;
   DATA[290,2] := 2.0;
   DATA[290,3] := 2.0;
   DATA[290,4] := 262.1764;
   DATA[290,5] := 8.39131;
   DATA[290,6] := 328.2492;
   DATA[290,7] := 2.442828;
   DATA[290,8] := 2.0;
   DATA[290,9] := 2.0;
   DATA[290,10] := 2.0;
   DATA[290,11] := 19.62674;
   DATA[290,12] := 2.211959;
   DATA[290,13] := 970.5444;
   DATA[290,14] := 1.0;
   DATA[290,15] := 2.0;
   DATA[290,16] := 1.0;
   DATA[290,17] := 1.0;
   DATA[290,18] := 1.0;
   DATA[290,19] := 2.0;
   DATA[290,20] := 148.808;
   DATA[290,21] := 156.0625;
   DATA[290,22] := 1.720437;
   DATA[290,23] := 965.9831;
   DATA[290,24] := 2.0;
   DATA[290,25] := 2.0;
   DATA[290,26] := 7.876058;
   DATA[290,27] := 144.8603;
   DATA[290,28] := 263.9067;
   DATA[290,29] := 12.11228;
   DATA[290,30] := 1.726865;
   DATA[290,31] := 1.311387;
   DATA[290,32] := 0.7351407;
   DATA[290,33] := 0.3065048;
   DATA[290,34] := 2.0;
   DATA[290,35] := 251.2657;
   DATA[290,36] := 1.649953;
   DATA[290,37] := 189.9353;
   DATA[290,38] := 0.000128152;
   DATA[290,39] := 1.0;
   DATA[291,0] := 2.656055;
   DATA[291,1] := 529.2449;
   DATA[291,2] := 2.0;
   DATA[291,3] := 2.0;
   DATA[291,4] := 262.1764;
   DATA[291,5] := 8.394514;
   DATA[291,6] := 328.2492;
   DATA[291,7] := 2.440137;
   DATA[291,8] := 2.0;
   DATA[291,9] := 2.0;
   DATA[291,10] := 2.0;
   DATA[291,11] := 19.58192;
   DATA[291,12] := 2.211959;
   DATA[291,13] := 970.224;
   DATA[291,14] := 1.0;
   DATA[291,15] := 2.0;
   DATA[291,16] := 1.0;
   DATA[291,17] := 1.0;
   DATA[291,18] := 1.0;
   DATA[291,19] := 2.0;
   DATA[291,20] := 148.808;
   DATA[291,21] := 156.0625;
   DATA[291,22] := 1.720437;
   DATA[291,23] := 966.0984;
   DATA[291,24] := 2.0;
   DATA[291,25] := 2.0;
   DATA[291,26] := 7.876058;
   DATA[291,27] := 144.8603;
   DATA[291,28] := 263.9067;
   DATA[291,29] := 12.11228;
   DATA[291,30] := 1.726865;
   DATA[291,31] := 1.303958;
   DATA[291,32] := 0.7351407;
   DATA[291,33] := 0.3065048;
   DATA[291,34] := 2.0;
   DATA[291,35] := 251.2657;
   DATA[291,36] := 1.826162;
   DATA[291,37] := 190.0634;
   DATA[291,38] := 0.000128152;
   DATA[291,39] := 1.0;
   DATA[292,0] := 2.670467;
   DATA[292,1] := 529.1664;
   DATA[292,2] := 2.0;
   DATA[292,3] := 2.0;
   DATA[292,4] := 262.1764;
   DATA[292,5] := 8.394514;
   DATA[292,6] := 328.2492;
   DATA[292,7] := 2.440137;
   DATA[292,8] := 2.0;
   DATA[292,9] := 2.0;
   DATA[292,10] := 2.0;
   DATA[292,11] := 19.57232;
   DATA[292,12] := 2.21119;
   DATA[292,13] := 970.224;
   DATA[292,14] := 1.0;
   DATA[292,15] := 2.0;
   DATA[292,16] := 1.0;
   DATA[292,17] := 1.0;
   DATA[292,18] := 1.0;
   DATA[292,19] := 2.0;
   DATA[292,20] := 148.808;
   DATA[292,21] := 156.0625;
   DATA[292,22] := 1.720437;
   DATA[292,23] := 965.9062;
   DATA[292,24] := 2.0;
   DATA[292,25] := 2.0;
   DATA[292,26] := 7.876058;
   DATA[292,27] := 144.8603;
   DATA[292,28] := 263.9067;
   DATA[292,29] := 12.11228;
   DATA[292,30] := 1.726865;
   DATA[292,31] := 1.291405;
   DATA[292,32] := 0.7351407;
   DATA[292,33] := 0.3065048;
   DATA[292,34] := 2.0;
   DATA[292,35] := 251.2657;
   DATA[292,36] := 1.826162;
   DATA[292,37] := 190.0634;
   DATA[292,38] := 0.000128152;
   DATA[292,39] := 1.0;
   DATA[293,0] := 2.671428;
   DATA[293,1] := 529.2057;
   DATA[293,2] := 2.0;
   DATA[293,3] := 2.0;
   DATA[293,4] := 262.1764;
   DATA[293,5] := 8.394514;
   DATA[293,6] := 328.2492;
   DATA[293,7] := 2.440137;
   DATA[293,8] := 2.0;
   DATA[293,9] := 2.0;
   DATA[293,10] := 2.0;
   DATA[293,11] := 19.61393;
   DATA[293,12] := 2.21119;
   DATA[293,13] := 970.0638;
   DATA[293,14] := 1.0;
   DATA[293,15] := 2.0;
   DATA[293,16] := 1.0;
   DATA[293,17] := 1.0;
   DATA[293,18] := 1.0;
   DATA[293,19] := 2.0;
   DATA[293,20] := 148.808;
   DATA[293,21] := 156.0625;
   DATA[293,22] := 1.719156;
   DATA[293,23] := 965.9831;
   DATA[293,24] := 2.0;
   DATA[293,25] := 2.0;
   DATA[293,26] := 7.876058;
   DATA[293,27] := 144.8603;
   DATA[293,28] := 263.9067;
   DATA[293,29] := 12.11228;
   DATA[293,30] := 1.727634;
   DATA[293,31] := 1.291405;
   DATA[293,32] := 0.7351407;
   DATA[293,33] := 0.3070813;
   DATA[293,34] := 2.0;
   DATA[293,35] := 251.2657;
   DATA[293,36] := 1.826162;
   DATA[293,37] := 190.0634;
   DATA[293,38] := 0.000128152;
   DATA[293,39] := 1.0;
   DATA[294,0] := 2.644845;
   DATA[294,1] := 529.4412;
   DATA[294,2] := 2.0;
   DATA[294,3] := 2.0;
   DATA[294,4] := 262.1764;
   DATA[294,5] := 8.394514;
   DATA[294,6] := 328.2492;
   DATA[294,7] := 2.441803;
   DATA[294,8] := 2.0;
   DATA[294,9] := 2.0;
   DATA[294,10] := 2.0;
   DATA[294,11] := 19.61393;
   DATA[294,12] := 2.212728;
   DATA[294,13] := 970.224;
   DATA[294,14] := 1.0;
   DATA[294,15] := 2.0;
   DATA[294,16] := 1.0;
   DATA[294,17] := 1.0;
   DATA[294,18] := 1.0;
   DATA[294,19] := 2.0;
   DATA[294,20] := 148.808;
   DATA[294,21] := 156.0625;
   DATA[294,22] := 1.717489;
   DATA[294,23] := 965.7139;
   DATA[294,24] := 2.0;
   DATA[294,25] := 2.0;
   DATA[294,26] := 7.876058;
   DATA[294,27] := 145.091;
   DATA[294,28] := 263.9067;
   DATA[294,29] := 12.07383;
   DATA[294,30] := 1.728788;
   DATA[294,31] := 1.291405;
   DATA[294,32] := 0.7351407;
   DATA[294,33] := 0.3070813;
   DATA[294,34] := 2.0;
   DATA[294,35] := 251.2657;
   DATA[294,36] := 1.681991;
   DATA[294,37] := 190.0634;
   DATA[294,38] := 0.000128152;
   DATA[294,39] := 1.0;
   DATA[295,0] := 2.625308;
   DATA[295,1] := 529.2449;
   DATA[295,2] := 2.0;
   DATA[295,3] := 2.0;
   DATA[295,4] := 262.1764;
   DATA[295,5] := 8.394514;
   DATA[295,6] := 328.2492;
   DATA[295,7] := 2.44206;
   DATA[295,8] := 2.0;
   DATA[295,9] := 2.0;
   DATA[295,10] := 2.0;
   DATA[295,11] := 19.61393;
   DATA[295,12] := 2.212728;
   DATA[295,13] := 970.0638;
   DATA[295,14] := 1.0;
   DATA[295,15] := 2.0;
   DATA[295,16] := 1.0;
   DATA[295,17] := 1.0;
   DATA[295,18] := 1.0;
   DATA[295,19] := 2.0;
   DATA[295,20] := 148.808;
   DATA[295,21] := 156.0625;
   DATA[295,22] := 1.717489;
   DATA[295,23] := 965.7139;
   DATA[295,24] := 2.0;
   DATA[295,25] := 2.0;
   DATA[295,26] := 7.876058;
   DATA[295,27] := 145.091;
   DATA[295,28] := 263.9067;
   DATA[295,29] := 12.07383;
   DATA[295,30] := 1.728788;
   DATA[295,31] := 1.300115;
   DATA[295,32] := 0.7351407;
   DATA[295,33] := 0.3070813;
   DATA[295,34] := 2.0;
   DATA[295,35] := 251.2657;
   DATA[295,36] := 1.681991;
   DATA[295,37] := 189.9032;
   DATA[295,38] := 0.000128152;
   DATA[295,39] := 1.0;
   DATA[296,0] := 2.621145;
   DATA[296,1] := 529.1272;
   DATA[296,2] := 2.0;
   DATA[296,3] := 2.0;
   DATA[296,4] := 262.1764;
   DATA[296,5] := 8.394514;
   DATA[296,6] := 328.2492;
   DATA[296,7] := 2.44206;
   DATA[296,8] := 2.0;
   DATA[296,9] := 2.0;
   DATA[296,10] := 2.0;
   DATA[296,11] := 19.61393;
   DATA[296,12] := 2.212728;
   DATA[296,13] := 969.6633;
   DATA[296,14] := 1.0;
   DATA[296,15] := 2.0;
   DATA[296,16] := 1.0;
   DATA[296,17] := 1.0;
   DATA[296,18] := 1.0;
   DATA[296,19] := 2.0;
   DATA[296,20] := 148.808;
   DATA[296,21] := 156.0625;
   DATA[296,22] := 1.717489;
   DATA[296,23] := 965.7524;
   DATA[296,24] := 2.0;
   DATA[296,25] := 2.0;
   DATA[296,26] := 7.877339;
   DATA[296,27] := 145.091;
   DATA[296,28] := 263.9067;
   DATA[296,29] := 12.07383;
   DATA[296,30] := 1.728788;
   DATA[296,31] := 1.292686;
   DATA[296,32] := 0.7351407;
   DATA[296,33] := 0.3066329;
   DATA[296,34] := 2.0;
   DATA[296,35] := 251.2657;
   DATA[296,36] := 1.681991;
   DATA[296,37] := 189.8552;
   DATA[296,38] := 0.000128152;
   DATA[296,39] := 1.0;
   DATA[297,0] := 2.616981;
   DATA[297,1] := 528.7347;
   DATA[297,2] := 2.0;
   DATA[297,3] := 2.0;
   DATA[297,4] := 262.1764;
   DATA[297,5] := 8.394514;
   DATA[297,6] := 328.2492;
   DATA[297,7] := 2.439496;
   DATA[297,8] := 2.0;
   DATA[297,9] := 2.0;
   DATA[297,10] := 2.0;
   DATA[297,11] := 19.63954;
   DATA[297,12] := 2.210166;
   DATA[297,13] := 969.4229;
   DATA[297,14] := 1.0;
   DATA[297,15] := 2.0;
   DATA[297,16] := 1.0;
   DATA[297,17] := 1.0;
   DATA[297,18] := 1.0;
   DATA[297,19] := 2.0;
   DATA[297,20] := 148.808;
   DATA[297,21] := 156.0625;
   DATA[297,22] := 1.717489;
   DATA[297,23] := 965.7139;
   DATA[297,24] := 2.0;
   DATA[297,25] := 2.0;
   DATA[297,26] := 7.877339;
   DATA[297,27] := 145.091;
   DATA[297,28] := 263.9067;
   DATA[297,29] := 12.07383;
   DATA[297,30] := 1.726096;
   DATA[297,31] := 1.281927;
   DATA[297,32] := 0.7351407;
   DATA[297,33] := 0.3066329;
   DATA[297,34] := 2.0;
   DATA[297,35] := 251.1055;
   DATA[297,36] := 1.681991;
   DATA[297,37] := 189.7751;
   DATA[297,38] := 0.000128152;
   DATA[297,39] := 1.0;
   DATA[298,0] := 2.602569;
   DATA[298,1] := 528.6169;
   DATA[298,2] := 2.0;
   DATA[298,3] := 2.0;
   DATA[298,4] := 262.1764;
   DATA[298,5] := 8.394514;
   DATA[298,6] := 328.0441;
   DATA[298,7] := 2.439496;
   DATA[298,8] := 2.0;
   DATA[298,9] := 2.0;
   DATA[298,10] := 2.0;
   DATA[298,11] := 19.73878;
   DATA[298,12] := 2.209525;
   DATA[298,13] := 969.3428;
   DATA[298,14] := 1.0;
   DATA[298,15] := 2.0;
   DATA[298,16] := 1.0;
   DATA[298,17] := 1.0;
   DATA[298,18] := 1.0;
   DATA[298,19] := 2.0;
   DATA[298,20] := 148.808;
   DATA[298,21] := 156.0625;
   DATA[298,22] := 1.717489;
   DATA[298,23] := 965.7139;
   DATA[298,24] := 2.0;
   DATA[298,25] := 2.0;
   DATA[298,26] := 7.877339;
   DATA[298,27] := 145.091;
   DATA[298,28] := 263.9067;
   DATA[298,29] := 12.07383;
   DATA[298,30] := 1.725711;
   DATA[298,31] := 1.278468;
   DATA[298,32] := 0.7351407;
   DATA[298,33] := 0.3066329;
   DATA[298,34] := 2.0;
   DATA[298,35] := 251.1055;
   DATA[298,36] := 1.681991;
   DATA[298,37] := 189.759;
   DATA[298,38] := 0.000128152;
   DATA[298,39] := 1.0;
   DATA[299,0] := 2.58079;
   DATA[299,1] := 528.2636;
   DATA[299,2] := 2.0;
   DATA[299,3] := 2.0;
   DATA[299,4] := 262.1764;
   DATA[299,5] := 8.394514;
   DATA[299,6] := 328.0441;
   DATA[299,7] := 2.439496;
   DATA[299,8] := 2.0;
   DATA[299,9] := 2.0;
   DATA[299,10] := 2.0;
   DATA[299,11] := 19.7804;
   DATA[299,12] := 2.209525;
   DATA[299,13] := 969.0624;
   DATA[299,14] := 1.0;
   DATA[299,15] := 2.0;
   DATA[299,16] := 1.0;
   DATA[299,17] := 1.0;
   DATA[299,18] := 1.0;
   DATA[299,19] := 2.0;
   DATA[299,20] := 148.808;
   DATA[299,21] := 156.0625;
   DATA[299,22] := 1.714029;
   DATA[299,23] := 965.5217;
   DATA[299,24] := 2.0;
   DATA[299,25] := 2.0;
   DATA[299,26] := 7.877339;
   DATA[299,27] := 144.8859;
   DATA[299,28] := 263.9067;
   DATA[299,29] := 12.07383;
   DATA[299,30] := 1.725711;
   DATA[299,31] := 1.268733;
   DATA[299,32] := 0.7351407;
   DATA[299,33] := 0.3066329;
   DATA[299,34] := 2.0;
   DATA[299,35] := 251.1055;
   DATA[299,36] := 1.681991;
   DATA[299,37] := 189.759;
   DATA[299,38] := 0.000128152;
   DATA[299,39] := 1.0;
   DATA[300,0] := 2.5699;
   DATA[300,1] := 528.2244;
   DATA[300,2] := 2.0;
   DATA[300,3] := 2.0;
   DATA[300,4] := 262.1764;
   DATA[300,5] := 8.394514;
   DATA[300,6] := 328.0441;
   DATA[300,7] := 2.439496;
   DATA[300,8] := 2.0;
   DATA[300,9] := 2.0;
   DATA[300,10] := 2.0;
   DATA[300,11] := 19.75799;
   DATA[300,12] := 2.209525;
   DATA[300,13] := 969.3428;
   DATA[300,14] := 1.0;
   DATA[300,15] := 2.0;
   DATA[300,16] := 1.0;
   DATA[300,17] := 1.0;
   DATA[300,18] := 1.0;
   DATA[300,19] := 2.0;
   DATA[300,20] := 148.808;
   DATA[300,21] := 155.9344;
   DATA[300,22] := 1.714029;
   DATA[300,23] := 965.6755;
   DATA[300,24] := 2.0;
   DATA[300,25] := 2.0;
   DATA[300,26] := 7.877339;
   DATA[300,27] := 144.8859;
   DATA[300,28] := 263.9067;
   DATA[300,29] := 12.07383;
   DATA[300,30] := 1.727634;
   DATA[300,31] := 1.261944;
   DATA[300,32] := 0.7351407;
   DATA[300,33] := 0.3066329;
   DATA[300,34] := 2.0;
   DATA[300,35] := 251.1055;
   DATA[300,36] := 1.681991;
   DATA[300,37] := 189.759;
   DATA[300,38] := 0.000128152;
   DATA[300,39] := 1.0;
   DATA[301,0] := 2.549082;
   DATA[301,1] := 528.3421;
   DATA[301,2] := 2.0;
   DATA[301,3] := 2.0;
   DATA[301,4] := 262.1764;
   DATA[301,5] := 8.394514;
   DATA[301,6] := 328.0441;
   DATA[301,7] := 2.439496;
   DATA[301,8] := 2.0;
   DATA[301,9] := 2.0;
   DATA[301,10] := 2.0;
   DATA[301,11] := 19.70677;
   DATA[301,12] := 2.209525;
   DATA[301,13] := 969.3428;
   DATA[301,14] := 1.0;
   DATA[301,15] := 2.0;
   DATA[301,16] := 1.0;
   DATA[301,17] := 1.0;
   DATA[301,18] := 1.0;
   DATA[301,19] := 2.0;
   DATA[301,20] := 148.808;
   DATA[301,21] := 155.9344;
   DATA[301,22] := 1.716721;
   DATA[301,23] := 966.06;
   DATA[301,24] := 2.0;
   DATA[301,25] := 2.0;
   DATA[301,26] := 7.877339;
   DATA[301,27] := 144.8859;
   DATA[301,28] := 263.9067;
   DATA[301,29] := 12.07383;
   DATA[301,30] := 1.728275;
   DATA[301,31] := 1.261944;
   DATA[301,32] := 0.7351407;
   DATA[301,33] := 0.3066329;
   DATA[301,34] := 2.0;
   DATA[301,35] := 251.1055;
   DATA[301,36] := 1.681991;
   DATA[301,37] := 189.759;
   DATA[301,38] := 0.000128152;
   DATA[301,39] := 1.0;
   DATA[302,0] := 2.535311;
   DATA[302,1] := 528.2636;
   DATA[302,2] := 2.0;
   DATA[302,3] := 2.0;
   DATA[302,4] := 262.1764;
   DATA[302,5] := 8.394514;
   DATA[302,6] := 328.0441;
   DATA[302,7] := 2.440521;
   DATA[302,8] := 2.0;
   DATA[302,9] := 2.0;
   DATA[302,10] := 2.0;
   DATA[302,11] := 19.70677;
   DATA[302,12] := 2.209525;
   DATA[302,13] := 969.5431;
   DATA[302,14] := 1.0;
   DATA[302,15] := 2.0;
   DATA[302,16] := 1.0;
   DATA[302,17] := 1.0;
   DATA[302,18] := 1.0;
   DATA[302,19] := 2.0;
   DATA[302,20] := 148.808;
   DATA[302,21] := 155.7806;
   DATA[302,22] := 1.717874;
   DATA[302,23] := 965.9062;
   DATA[302,24] := 2.0;
   DATA[302,25] := 2.0;
   DATA[302,26] := 7.877339;
   DATA[302,27] := 144.8859;
   DATA[302,28] := 263.9067;
   DATA[302,29] := 12.07383;
   DATA[302,30] := 1.728275;
   DATA[302,31] := 1.261944;
   DATA[302,32] := 0.7351407;
   DATA[302,33] := 0.3066329;
   DATA[302,34] := 2.0;
   DATA[302,35] := 251.1055;
   DATA[302,36] := 1.681991;
   DATA[302,37] := 189.759;
   DATA[302,38] := 0.000128152;
   DATA[302,39] := 1.0;
   DATA[303,0] := 2.518336;
   DATA[303,1] := 528.2244;
   DATA[303,2] := 2.0;
   DATA[303,3] := 2.0;
   DATA[303,4] := 262.1764;
   DATA[303,5] := 8.394514;
   DATA[303,6] := 328.0441;
   DATA[303,7] := 2.440521;
   DATA[303,8] := 2.0;
   DATA[303,9] := 2.0;
   DATA[303,10] := 2.0;
   DATA[303,11] := 19.70677;
   DATA[303,12] := 2.209525;
   DATA[303,13] := 969.9837;
   DATA[303,14] := 1.0;
   DATA[303,15] := 2.0;
   DATA[303,16] := 1.0;
   DATA[303,17] := 1.0;
   DATA[303,18] := 1.0;
   DATA[303,19] := 2.0;
   DATA[303,20] := 148.808;
   DATA[303,21] := 155.7293;
   DATA[303,22] := 1.719284;
   DATA[303,23] := 965.5986;
   DATA[303,24] := 2.0;
   DATA[303,25] := 2.0;
   DATA[303,26] := 7.877339;
   DATA[303,27] := 144.8859;
   DATA[303,28] := 263.9067;
   DATA[303,29] := 12.07383;
   DATA[303,30] := 1.728788;
   DATA[303,31] := 1.261944;
   DATA[303,32] := 0.7351407;
   DATA[303,33] := 0.3066329;
   DATA[303,34] := 2.0;
   DATA[303,35] := 251.1055;
   DATA[303,36] := 1.681991;
   DATA[303,37] := 189.759;
   DATA[303,38] := 0.000128152;
   DATA[303,39] := 1.0;
   DATA[304,0] := 2.503923;
   DATA[304,1] := 528.3421;
   DATA[304,2] := 2.0;
   DATA[304,3] := 2.0;
   DATA[304,4] := 262.1764;
   DATA[304,5] := 8.394514;
   DATA[304,6] := 328.0441;
   DATA[304,7] := 2.441803;
   DATA[304,8] := 2.0;
   DATA[304,9] := 2.0;
   DATA[304,10] := 2.0;
   DATA[304,11] := 19.70677;
   DATA[304,12] := 2.209525;
   DATA[304,13] := 969.9436;
   DATA[304,14] := 1.0;
   DATA[304,15] := 2.0;
   DATA[304,16] := 1.0;
   DATA[304,17] := 1.0;
   DATA[304,18] := 1.0;
   DATA[304,19] := 2.0;
   DATA[304,20] := 148.808;
   DATA[304,21] := 155.7293;
   DATA[304,22] := 1.719284;
   DATA[304,23] := 965.7908;
   DATA[304,24] := 2.0;
   DATA[304,25] := 2.0;
   DATA[304,26] := 7.877339;
   DATA[304,27] := 145.0141;
   DATA[304,28] := 263.9067;
   DATA[304,29] := 12.07383;
   DATA[304,30] := 1.728788;
   DATA[304,31] := 1.271423;
   DATA[304,32] := 0.7351407;
   DATA[304,33] := 0.3066329;
   DATA[304,34] := 2.0;
   DATA[304,35] := 251.1055;
   DATA[304,36] := 1.681991;
   DATA[304,37] := 189.759;
   DATA[304,38] := 0.000128152;
   DATA[304,39] := 1.0;
   DATA[305,0] := 2.484386;
   DATA[305,1] := 528.7347;
   DATA[305,2] := 2.0;
   DATA[305,3] := 2.0;
   DATA[305,4] := 262.1764;
   DATA[305,5] := 8.394514;
   DATA[305,6] := 328.0954;
   DATA[305,7] := 2.442188;
   DATA[305,8] := 2.0;
   DATA[305,9] := 2.0;
   DATA[305,10] := 2.0;
   DATA[305,11] := 19.74198;
   DATA[305,12] := 2.209525;
   DATA[305,13] := 970.224;
   DATA[305,14] := 1.0;
   DATA[305,15] := 2.0;
   DATA[305,16] := 1.0;
   DATA[305,17] := 1.0;
   DATA[305,18] := 1.0;
   DATA[305,19] := 2.0;
   DATA[305,20] := 148.808;
   DATA[305,21] := 155.7293;
   DATA[305,22] := 1.718387;
   DATA[305,23] := 965.6755;
   DATA[305,24] := 2.0;
   DATA[305,25] := 2.0;
   DATA[305,26] := 7.877339;
   DATA[305,27] := 145.0141;
   DATA[305,28] := 263.9067;
   DATA[305,29] := 12.07383;
   DATA[305,30] := 1.728788;
   DATA[305,31] := 1.276803;
   DATA[305,32] := 0.7351407;
   DATA[305,33] := 0.3066329;
   DATA[305,34] := 2.0;
   DATA[305,35] := 251.1055;
   DATA[305,36] := 1.681991;
   DATA[305,37] := 189.759;
   DATA[305,38] := 0.000128152;
   DATA[305,39] := 1.0;
   DATA[306,0] := 2.472857;
   DATA[306,1] := 528.4599;
   DATA[306,2] := 2.0;
   DATA[306,3] := 2.0;
   DATA[306,4] := 262.1764;
   DATA[306,5] := 8.394514;
   DATA[306,6] := 328.2492;
   DATA[306,7] := 2.442188;
   DATA[306,8] := 2.0;
   DATA[306,9] := 2.0;
   DATA[306,10] := 2.0;
   DATA[306,11] := 19.74198;
   DATA[306,12] := 2.209525;
   DATA[306,13] := 970.0638;
   DATA[306,14] := 1.0;
   DATA[306,15] := 2.0;
   DATA[306,16] := 1.0;
   DATA[306,17] := 1.0;
   DATA[306,18] := 1.0;
   DATA[306,19] := 2.0;
   DATA[306,20] := 148.808;
   DATA[306,21] := 155.7293;
   DATA[306,22] := 1.716849;
   DATA[306,23] := 966.06;
   DATA[306,24] := 2.0;
   DATA[306,25] := 2.0;
   DATA[306,26] := 7.879582;
   DATA[306,27] := 145.0141;
   DATA[306,28] := 263.9067;
   DATA[306,29] := 12.26609;
   DATA[306,30] := 1.728788;
   DATA[306,31] := 1.281286;
   DATA[306,32] := 0.7351407;
   DATA[306,33] := 0.3066329;
   DATA[306,34] := 2.0;
   DATA[306,35] := 251.1055;
   DATA[306,36] := 1.810143;
   DATA[306,37] := 189.759;
   DATA[306,38] := 0.000128152;
   DATA[306,39] := 1.0;
   DATA[307,0] := 2.457163;
   DATA[307,1] := 528.3421;
   DATA[307,2] := 2.0;
   DATA[307,3] := 2.0;
   DATA[307,4] := 262.1764;
   DATA[307,5] := 8.394514;
   DATA[307,6] := 328.2492;
   DATA[307,7] := 2.442188;
   DATA[307,8] := 2.0;
   DATA[307,9] := 2.0;
   DATA[307,10] := 2.0;
   DATA[307,11] := 19.74198;
   DATA[307,12] := 2.209525;
   DATA[307,13] := 970.3842;
   DATA[307,14] := 1.0;
   DATA[307,15] := 2.0;
   DATA[307,16] := 1.0;
   DATA[307,17] := 1.0;
   DATA[307,18] := 1.0;
   DATA[307,19] := 2.0;
   DATA[307,20] := 148.808;
   DATA[307,21] := 155.7293;
   DATA[307,22] := 1.716849;
   DATA[307,23] := 966.5214;
   DATA[307,24] := 2.0;
   DATA[307,25] := 2.0;
   DATA[307,26] := 7.879582;
   DATA[307,27] := 145.0141;
   DATA[307,28] := 263.9067;
   DATA[307,29] := 12.26609;
   DATA[307,30] := 1.728788;
   DATA[307,31] := 1.268349;
   DATA[307,32] := 0.7351407;
   DATA[307,33] := 0.3066329;
   DATA[307,34] := 2.0;
   DATA[307,35] := 251.1055;
   DATA[307,36] := 1.810143;
   DATA[307,37] := 189.759;
   DATA[307,38] := 0.000128152;
   DATA[307,39] := 1.0;
   DATA[308,0] := 2.445633;
   DATA[308,1] := 528.5384;
   DATA[308,2] := 2.0;
   DATA[308,3] := 2.0;
   DATA[308,4] := 262.1764;
   DATA[308,5] := 8.39163;
   DATA[308,6] := 328.2492;
   DATA[308,7] := 2.442188;
   DATA[308,8] := 2.0;
   DATA[308,9] := 2.0;
   DATA[308,10] := 2.0;
   DATA[308,11] := 19.74198;
   DATA[308,12] := 2.209525;
   DATA[308,13] := 970.4243;
   DATA[308,14] := 1.0;
   DATA[308,15] := 2.0;
   DATA[308,16] := 1.0;
   DATA[308,17] := 1.0;
   DATA[308,18] := 1.0;
   DATA[308,19] := 2.0;
   DATA[308,20] := 148.808;
   DATA[308,21] := 155.6524;
   DATA[308,22] := 1.716849;
   DATA[308,23] := 966.4445;
   DATA[308,24] := 2.0;
   DATA[308,25] := 2.0;
   DATA[308,26] := 7.879582;
   DATA[308,27] := 145.0141;
   DATA[308,28] := 263.9067;
   DATA[308,29] := 12.26609;
   DATA[308,30] := 1.728788;
   DATA[308,31] := 1.261944;
   DATA[308,32] := 0.7351407;
   DATA[308,33] := 0.3066329;
   DATA[308,34] := 2.0;
   DATA[308,35] := 251.1055;
   DATA[308,36] := 1.810143;
   DATA[308,37] := 189.759;
   DATA[308,38] := 0.000128152;
   DATA[308,39] := 1.0;
   DATA[309,0] := 2.431541;
   DATA[309,1] := 528.7347;
   DATA[309,2] := 2.0;
   DATA[309,3] := 2.0;
   DATA[309,4] := 262.1764;
   DATA[309,5] := 8.39163;
   DATA[309,6] := 328.2492;
   DATA[309,7] := 2.440137;
   DATA[309,8] := 2.0;
   DATA[309,9] := 2.0;
   DATA[309,10] := 2.0;
   DATA[309,11] := 19.74198;
   DATA[309,12] := 2.210294;
   DATA[309,13] := 970.6646;
   DATA[309,14] := 1.0;
   DATA[309,15] := 2.0;
   DATA[309,16] := 1.0;
   DATA[309,17] := 1.0;
   DATA[309,18] := 1.0;
   DATA[309,19] := 2.0;
   DATA[309,20] := 148.808;
   DATA[309,21] := 155.6524;
   DATA[309,22] := 1.716849;
   DATA[309,23] := 966.2907;
   DATA[309,24] := 2.0;
   DATA[309,25] := 2.0;
   DATA[309,26] := 7.879582;
   DATA[309,27] := 145.0141;
   DATA[309,28] := 263.9067;
   DATA[309,29] := 12.26609;
   DATA[309,30] := 1.726865;
   DATA[309,31] := 1.253362;
   DATA[309,32] := 0.7351407;
   DATA[309,33] := 0.3066329;
   DATA[309,34] := 2.0;
   DATA[309,35] := 251.1055;
   DATA[309,36] := 1.810143;
   DATA[309,37] := 189.759;
   DATA[309,38] := 0.000128152;
   DATA[309,39] := 1.0;
   DATA[310,0] := 2.423534;
   DATA[310,1] := 528.8132;
   DATA[310,2] := 2.0;
   DATA[310,3] := 2.0;
   DATA[310,4] := 262.1764;
   DATA[310,5] := 8.39163;
   DATA[310,6] := 328.2492;
   DATA[310,7] := 2.440137;
   DATA[310,8] := 2.0;
   DATA[310,9] := 2.0;
   DATA[310,10] := 2.0;
   DATA[310,11] := 19.72598;
   DATA[310,12] := 2.212087;
   DATA[310,13] := 970.7447;
   DATA[310,14] := 1.0;
   DATA[310,15] := 2.0;
   DATA[310,16] := 1.0;
   DATA[310,17] := 1.0;
   DATA[310,18] := 1.0;
   DATA[310,19] := 2.0;
   DATA[310,20] := 148.808;
   DATA[310,21] := 155.6524;
   DATA[310,22] := 1.716849;
   DATA[310,23] := 966.7521;
   DATA[310,24] := 2.0;
   DATA[310,25] := 2.0;
   DATA[310,26] := 7.879582;
   DATA[310,27] := 145.0141;
   DATA[310,28] := 263.9067;
   DATA[310,29] := 11.88157;
   DATA[310,30] := 1.726737;
   DATA[310,31] := 1.246189;
   DATA[310,32] := 0.7351407;
   DATA[310,33] := 0.3070813;
   DATA[310,34] := 2.0;
   DATA[310,35] := 251.1055;
   DATA[310,36] := 1.69801;
   DATA[310,37] := 189.759;
   DATA[310,38] := 0.000128152;
   DATA[310,39] := 1.0;
   DATA[311,0] := 2.423534;
   DATA[311,1] := 528.8524;
   DATA[311,2] := 2.0;
   DATA[311,3] := 2.0;
   DATA[311,4] := 262.1764;
   DATA[311,5] := 8.39163;
   DATA[311,6] := 328.2492;
   DATA[311,7] := 2.440137;
   DATA[311,8] := 2.0;
   DATA[311,9] := 2.0;
   DATA[311,10] := 2.0;
   DATA[311,11] := 19.72598;
   DATA[311,12] := 2.212087;
   DATA[311,13] := 970.6646;
   DATA[311,14] := 1.0;
   DATA[311,15] := 2.0;
   DATA[311,16] := 1.0;
   DATA[311,17] := 1.0;
   DATA[311,18] := 1.0;
   DATA[311,19] := 2.0;
   DATA[311,20] := 148.808;
   DATA[311,21] := 155.6524;
   DATA[311,22] := 1.716849;
   DATA[311,23] := 967.1367;
   DATA[311,24] := 2.0;
   DATA[311,25] := 2.0;
   DATA[311,26] := 7.879582;
   DATA[311,27] := 145.2448;
   DATA[311,28] := 263.9067;
   DATA[311,29] := 11.88157;
   DATA[311,30] := 1.726224;
   DATA[311,31] := 1.259383;
   DATA[311,32] := 0.7351407;
   DATA[311,33] := 0.3070813;
   DATA[311,34] := 2.0;
   DATA[311,35] := 251.1055;
   DATA[311,36] := 1.69801;
   DATA[311,37] := 189.759;
   DATA[311,38] := 0.000128152;
   DATA[311,39] := 1.0;
   DATA[312,0] := 2.439868;
   DATA[312,1] := 528.8132;
   DATA[312,2] := 2.0;
   DATA[312,3] := 2.0;
   DATA[312,4] := 262.1764;
   DATA[312,5] := 8.39163;
   DATA[312,6] := 328.2492;
   DATA[312,7] := 2.440137;
   DATA[312,8] := 2.0;
   DATA[312,9] := 2.0;
   DATA[312,10] := 2.0;
   DATA[312,11] := 19.7996;
   DATA[312,12] := 2.212087;
   DATA[312,13] := 970.9449;
   DATA[312,14] := 1.0;
   DATA[312,15] := 2.0;
   DATA[312,16] := 1.0;
   DATA[312,17] := 1.0;
   DATA[312,18] := 1.0;
   DATA[312,19] := 2.0;
   DATA[312,20] := 148.808;
   DATA[312,21] := 155.6524;
   DATA[312,22] := 1.716849;
   DATA[312,23] := 967.1367;
   DATA[312,24] := 2.0;
   DATA[312,25] := 2.0;
   DATA[312,26] := 7.879582;
   DATA[312,27] := 145.2448;
   DATA[312,28] := 263.9067;
   DATA[312,29] := 12.15073;
   DATA[312,30] := 1.726224;
   DATA[312,31] := 1.270398;
   DATA[312,32] := 0.7351407;
   DATA[312,33] := 0.3070813;
   DATA[312,34] := 2.0;
   DATA[312,35] := 251.1055;
   DATA[312,36] := 1.69801;
   DATA[312,37] := 189.759;
   DATA[312,38] := 0.000128152;
   DATA[312,39] := 1.0;
   DATA[313,0] := 2.479582;
   DATA[313,1] := 528.7739;
   DATA[313,2] := 2.0;
   DATA[313,3] := 2.0;
   DATA[313,4] := 262.1764;
   DATA[313,5] := 8.39163;
   DATA[313,6] := 328.2492;
   DATA[313,7] := 2.440137;
   DATA[313,8] := 2.0;
   DATA[313,9] := 2.0;
   DATA[313,10] := 2.0;
   DATA[313,11] := 19.7996;
   DATA[313,12] := 2.212087;
   DATA[313,13] := 971.2253;
   DATA[313,14] := 1.0;
   DATA[313,15] := 2.0;
   DATA[313,16] := 1.0;
   DATA[313,17] := 1.0;
   DATA[313,18] := 1.0;
   DATA[313,19] := 2.0;
   DATA[313,20] := 148.808;
   DATA[313,21] := 155.6524;
   DATA[313,22] := 1.716849;
   DATA[313,23] := 967.598;
   DATA[313,24] := 2.0;
   DATA[313,25] := 2.0;
   DATA[313,26] := 7.879582;
   DATA[313,27] := 145.2192;
   DATA[313,28] := 263.9067;
   DATA[313,29] := 12.15073;
   DATA[313,30] := 1.726224;
   DATA[313,31] := 1.270911;
   DATA[313,32] := 0.7351407;
   DATA[313,33] := 0.3070813;
   DATA[313,34] := 2.0;
   DATA[313,35] := 250.9453;
   DATA[313,36] := 1.69801;
   DATA[313,37] := 189.759;
   DATA[313,38] := 0.000128152;
   DATA[313,39] := 1.0;
   DATA[314,0] := 2.520257;
   DATA[314,1] := 528.9702;
   DATA[314,2] := 2.0;
   DATA[314,3] := 2.0;
   DATA[314,4] := 262.0802;
   DATA[314,5] := 8.39163;
   DATA[314,6] := 328.2492;
   DATA[314,7] := 2.440137;
   DATA[314,8] := 2.0;
   DATA[314,9] := 2.0;
   DATA[314,10] := 2.0;
   DATA[314,11] := 19.7996;
   DATA[314,12] := 2.212087;
   DATA[314,13] := 971.3455;
   DATA[314,14] := 1.0;
   DATA[314,15] := 2.0;
   DATA[314,16] := 1.0;
   DATA[314,17] := 1.0;
   DATA[314,18] := 1.0;
   DATA[314,19] := 2.0;
   DATA[314,20] := 148.808;
   DATA[314,21] := 155.6524;
   DATA[314,22] := 1.717233;
   DATA[314,23] := 967.8287;
   DATA[314,24] := 2.0;
   DATA[314,25] := 2.0;
   DATA[314,26] := 7.879582;
   DATA[314,27] := 145.2192;
   DATA[314,28] := 263.9067;
   DATA[314,29] := 12.15073;
   DATA[314,30] := 1.726609;
   DATA[314,31] := 1.266556;
   DATA[314,32] := 0.7351407;
   DATA[314,33] := 0.3086827;
   DATA[314,34] := 2.0;
   DATA[314,35] := 250.9453;
   DATA[314,36] := 1.69801;
   DATA[314,37] := 189.759;
   DATA[314,38] := 0.000128152;
   DATA[314,39] := 1.0;
   DATA[315,0] := 2.561573;
   DATA[315,1] := 529.1272;
   DATA[315,2] := 2.0;
   DATA[315,3] := 2.0;
   DATA[315,4] := 262.0482;
   DATA[315,5] := 8.39163;
   DATA[315,6] := 328.1723;
   DATA[315,7] := 2.440137;
   DATA[315,8] := 2.0;
   DATA[315,9] := 2.0;
   DATA[315,10] := 2.0;
   DATA[315,11] := 19.7996;
   DATA[315,12] := 2.212343;
   DATA[315,13] := 971.4256;
   DATA[315,14] := 1.0;
   DATA[315,15] := 2.0;
   DATA[315,16] := 1.0;
   DATA[315,17] := 1.0;
   DATA[315,18] := 1.0;
   DATA[315,19] := 2.0;
   DATA[315,20] := 148.808;
   DATA[315,21] := 155.6524;
   DATA[315,22] := 1.717233;
   DATA[315,23] := 968.0979;
   DATA[315,24] := 2.0;
   DATA[315,25] := 2.0;
   DATA[315,26] := 7.879262;
   DATA[315,27] := 145.2192;
   DATA[315,28] := 263.9067;
   DATA[315,29] := 12.15073;
   DATA[315,30] := 1.726865;
   DATA[315,31] := 1.271679;
   DATA[315,32] := 0.7361649;
   DATA[315,33] := 0.3086827;
   DATA[315,34] := 2.0;
   DATA[315,35] := 250.8331;
   DATA[315,36] := 1.69801;
   DATA[315,37] := 189.759;
   DATA[315,38] := 0.000128152;
   DATA[315,39] := 1.0;
   DATA[316,0] := 2.595522;
   DATA[316,1] := 529.1272;
   DATA[316,2] := 2.0;
   DATA[316,3] := 2.0;
   DATA[316,4] := 262.0482;
   DATA[316,5] := 8.394514;
   DATA[316,6] := 328.0954;
   DATA[316,7] := 2.440137;
   DATA[316,8] := 2.0;
   DATA[316,9] := 2.0;
   DATA[316,10] := 2.0;
   DATA[316,11] := 19.7996;
   DATA[316,12] := 2.21324;
   DATA[316,13] := 971.0251;
   DATA[316,14] := 1.0;
   DATA[316,15] := 2.0;
   DATA[316,16] := 1.0;
   DATA[316,17] := 1.0;
   DATA[316,18] := 1.0;
   DATA[316,19] := 2.0;
   DATA[316,20] := 148.808;
   DATA[316,21] := 155.6524;
   DATA[316,22] := 1.717233;
   DATA[316,23] := 968.2517;
   DATA[316,24] := 2.0;
   DATA[316,25] := 2.0;
   DATA[316,26] := 7.878942;
   DATA[316,27] := 144.9628;
   DATA[316,28] := 263.9067;
   DATA[316,29] := 12.07383;
   DATA[316,30] := 1.726865;
   DATA[316,31] := 1.283079;
   DATA[316,32] := 0.7361649;
   DATA[316,33] := 0.3086827;
   DATA[316,34] := 2.0;
   DATA[316,35] := 250.6248;
   DATA[316,36] := 1.69801;
   DATA[316,37] := 189.6148;
   DATA[316,38] := 0.000128152;
   DATA[316,39] := 1.0;
   DATA[317,0] := 2.625949;
   DATA[317,1] := 529.1664;
   DATA[317,2] := 2.0;
   DATA[317,3] := 2.0;
   DATA[317,4] := 262.0482;
   DATA[317,5] := 8.396437;
   DATA[317,6] := 328.0441;
   DATA[317,7] := 2.440137;
   DATA[317,8] := 2.0;
   DATA[317,9] := 2.0;
   DATA[317,10] := 2.0;
   DATA[317,11] := 19.7996;
   DATA[317,12] := 2.21324;
   DATA[317,13] := 970.9449;
   DATA[317,14] := 1.0;
   DATA[317,15] := 2.0;
   DATA[317,16] := 1.0;
   DATA[317,17] := 1.0;
   DATA[317,18] := 1.0;
   DATA[317,19] := 2.0;
   DATA[317,20] := 148.808;
   DATA[317,21] := 155.6524;
   DATA[317,22] := 1.715439;
   DATA[317,23] := 968.5593;
   DATA[317,24] := 2.0;
   DATA[317,25] := 2.0;
   DATA[317,26] := 7.878942;
   DATA[317,27] := 144.9628;
   DATA[317,28] := 263.9067;
   DATA[317,29] := 12.03538;
   DATA[317,30] := 1.726865;
   DATA[317,31] := 1.298962;
   DATA[317,32] := 0.7361649;
   DATA[317,33] := 0.3086827;
   DATA[317,34] := 2.0;
   DATA[317,35] := 250.6248;
   DATA[317,36] := 1.69801;
   DATA[317,37] := 189.5027;
   DATA[317,38] := 0.000128152;
   DATA[317,39] := 1.0;
   DATA[318,0] := 2.647727;
   DATA[318,1] := 528.9702;
   DATA[318,2] := 2.0;
   DATA[318,3] := 2.0;
   DATA[318,4] := 262.0482;
   DATA[318,5] := 8.396437;
   DATA[318,6] := 328.0441;
   DATA[318,7] := 2.440137;
   DATA[318,8] := 2.0;
   DATA[318,9] := 2.0;
   DATA[318,10] := 2.0;
   DATA[318,11] := 19.7996;
   DATA[318,12] := 2.210934;
   DATA[318,13] := 970.6245;
   DATA[318,14] := 1.0;
   DATA[318,15] := 2.0;
   DATA[318,16] := 1.0;
   DATA[318,17] := 1.0;
   DATA[318,18] := 1.0;
   DATA[318,19] := 2.0;
   DATA[318,20] := 148.808;
   DATA[318,21] := 155.6524;
   DATA[318,22] := 1.715439;
   DATA[318,23] := 968.8285;
   DATA[318,24] := 2.0;
   DATA[318,25] := 2.0;
   DATA[318,26] := 7.878942;
   DATA[318,27] := 144.9628;
   DATA[318,28] := 263.9067;
   DATA[318,29] := 12.03538;
   DATA[318,30] := 1.726865;
   DATA[318,31] := 1.302165;
   DATA[318,32] := 0.7361649;
   DATA[318,33] := 0.3086827;
   DATA[318,34] := 2.0;
   DATA[318,35] := 250.6248;
   DATA[318,36] := 1.69801;
   DATA[318,37] := 189.4867;
   DATA[318,38] := 0.000128152;
   DATA[318,39] := 1.0;
   DATA[319,0] := 2.654453;
   DATA[319,1] := 528.6169;
   DATA[319,2] := 2.0;
   DATA[319,3] := 2.0;
   DATA[319,4] := 262.0482;
   DATA[319,5] := 8.396437;
   DATA[319,6] := 328.0441;
   DATA[319,7] := 2.440137;
   DATA[319,8] := 2.0;
   DATA[319,9] := 2.0;
   DATA[319,10] := 2.0;
   DATA[319,11] := 19.7996;
   DATA[319,12] := 2.21055;
   DATA[319,13] := 970.9449;
   DATA[319,14] := 1.0;
   DATA[319,15] := 2.0;
   DATA[319,16] := 1.0;
   DATA[319,17] := 1.0;
   DATA[319,18] := 1.0;
   DATA[319,19] := 2.0;
   DATA[319,20] := 148.808;
   DATA[319,21] := 155.6524;
   DATA[319,22] := 1.715439;
   DATA[319,23] := 968.9438;
   DATA[319,24] := 2.0;
   DATA[319,25] := 2.0;
   DATA[319,26] := 7.878942;
   DATA[319,27] := 145.0397;
   DATA[319,28] := 263.9067;
   DATA[319,29] := 12.03538;
   DATA[319,30] := 1.726865;
   DATA[319,31] := 1.302165;
   DATA[319,32] := 0.7352687;
   DATA[319,33] := 0.3084265;
   DATA[319,34] := 2.0;
   DATA[319,35] := 250.785;
   DATA[319,36] := 1.69801;
   DATA[319,37] := 189.4867;
   DATA[319,38] := 0.000128152;
   DATA[319,39] := 1.0;
   DATA[320,0] := 2.647727;
   DATA[320,1] := 528.2244;
   DATA[320,2] := 2.0;
   DATA[320,3] := 2.0;
   DATA[320,4] := 262.0482;
   DATA[320,5] := 8.393873;
   DATA[320,6] := 328.0441;
   DATA[320,7] := 2.440137;
   DATA[320,8] := 2.0;
   DATA[320,9] := 2.0;
   DATA[320,10] := 2.0;
   DATA[320,11] := 19.7996;
   DATA[320,12] := 2.209269;
   DATA[320,13] := 971.2654;
   DATA[320,14] := 1.0;
   DATA[320,15] := 2.0;
   DATA[320,16] := 1.0;
   DATA[320,17] := 1.0;
   DATA[320,18] := 1.0;
   DATA[320,19] := 2.0;
   DATA[320,20] := 148.808;
   DATA[320,21] := 155.6524;
   DATA[320,22] := 1.713901;
   DATA[320,23] := 969.3284;
   DATA[320,24] := 2.0;
   DATA[320,25] := 2.0;
   DATA[320,26] := 7.878942;
   DATA[320,27] := 145.0397;
   DATA[320,28] := 263.9067;
   DATA[320,29] := 12.03538;
   DATA[320,30] := 1.726737;
   DATA[320,31] := 1.29845;
   DATA[320,32] := 0.7352687;
   DATA[320,33] := 0.3079781;
   DATA[320,34] := 2.0;
   DATA[320,35] := 250.9132;
   DATA[320,36] := 1.69801;
   DATA[320,37] := 189.4867;
   DATA[320,38] := 0.000128152;
   DATA[320,39] := 1.0;
   DATA[321,0] := 2.63844;
   DATA[321,1] := 527.7534;
   DATA[321,2] := 2.0;
   DATA[321,3] := 2.0;
   DATA[321,4] := 262.0482;
   DATA[321,5] := 8.393873;
   DATA[321,6] := 328.0441;
   DATA[321,7] := 2.440137;
   DATA[321,8] := 2.0;
   DATA[321,9] := 2.0;
   DATA[321,10] := 2.0;
   DATA[321,11] := 19.77399;
   DATA[321,12] := 2.209269;
   DATA[321,13] := 971.0651;
   DATA[321,14] := 1.0;
   DATA[321,15] := 2.0;
   DATA[321,16] := 1.0;
   DATA[321,17] := 1.0;
   DATA[321,18] := 1.0;
   DATA[321,19] := 2.0;
   DATA[321,20] := 148.808;
   DATA[321,21] := 155.6524;
   DATA[321,22] := 1.712876;
   DATA[321,23] := 969.5591;
   DATA[321,24] := 2.0;
   DATA[321,25] := 2.0;
   DATA[321,26] := 7.878942;
   DATA[321,27] := 145.1166;
   DATA[321,28] := 263.9067;
   DATA[321,29] := 12.03538;
   DATA[321,30] := 1.726096;
   DATA[321,31] := 1.292558;
   DATA[321,32] := 0.7352687;
   DATA[321,33] := 0.3079781;
   DATA[321,34] := 2.0;
   DATA[321,35] := 250.9132;
   DATA[321,36] := 1.69801;
   DATA[321,37] := 189.5027;
   DATA[321,38] := 0.000128152;
   DATA[321,39] := 1.0;
   DATA[322,0] := 2.620824;
   DATA[322,1] := 527.2823;
   DATA[322,2] := 2.0;
   DATA[322,3] := 2.0;
   DATA[322,4] := 262.0482;
   DATA[322,5] := 8.393553;
   DATA[322,6] := 328.1723;
   DATA[322,7] := 2.440137;
   DATA[322,8] := 2.0;
   DATA[322,9] := 2.0;
   DATA[322,10] := 2.0;
   DATA[322,11] := 19.76759;
   DATA[322,12] := 2.209269;
   DATA[322,13] := 971.0251;
   DATA[322,14] := 1.0;
   DATA[322,15] := 2.0;
   DATA[322,16] := 1.0;
   DATA[322,17] := 1.0;
   DATA[322,18] := 1.0;
   DATA[322,19] := 2.0;
   DATA[322,20] := 148.808;
   DATA[322,21] := 155.6524;
   DATA[322,22] := 1.712748;
   DATA[322,23] := 969.9436;
   DATA[322,24] := 2.0;
   DATA[322,25] := 2.0;
   DATA[322,26] := 7.878942;
   DATA[322,27] := 145.1679;
   DATA[322,28] := 263.9067;
   DATA[322,29] := 12.03538;
   DATA[322,30] := 1.725455;
   DATA[322,31] := 1.288331;
   DATA[322,32] := 0.7352687;
   DATA[322,33] := 0.3079781;
   DATA[322,34] := 2.0;
   DATA[322,35] := 250.9132;
   DATA[322,36] := 1.69801;
   DATA[322,37] := 189.5988;
   DATA[322,38] := 0.000128152;
   DATA[322,39] := 1.0;
   DATA[323,0] := 2.617301;
   DATA[323,1] := 527.0075;
   DATA[323,2] := 2.0;
   DATA[323,3] := 2.0;
   DATA[323,4] := 262.0482;
   DATA[323,5] := 8.393553;
   DATA[323,6] := 328.1723;
   DATA[323,7] := 2.440137;
   DATA[323,8] := 2.0;
   DATA[323,9] := 2.0;
   DATA[323,10] := 2.0;
   DATA[323,11] := 19.76759;
   DATA[323,12] := 2.209269;
   DATA[323,13] := 971.5458;
   DATA[323,14] := 1.0;
   DATA[323,15] := 2.0;
   DATA[323,16] := 1.0;
   DATA[323,17] := 1.0;
   DATA[323,18] := 1.0;
   DATA[323,19] := 2.0;
   DATA[323,20] := 148.808;
   DATA[323,21] := 155.6524;
   DATA[323,22] := 1.714158;
   DATA[323,23] := 970.5973;
   DATA[323,24] := 2.0;
   DATA[323,25] := 2.0;
   DATA[323,26] := 7.878942;
   DATA[323,27] := 145.1679;
   DATA[323,28] := 263.9067;
   DATA[323,29] := 12.03538;
   DATA[323,30] := 1.725455;
   DATA[323,31] := 1.27834;
   DATA[323,32] := 0.7352687;
   DATA[323,33] := 0.3064407;
   DATA[323,34] := 2.0;
   DATA[323,35] := 250.9132;
   DATA[323,36] := 1.69801;
   DATA[323,37] := 189.5988;
   DATA[323,38] := 0.000128152;
   DATA[323,39] := 1.0;
   DATA[324,0] := 2.60481;
   DATA[324,1] := 527.243;
   DATA[324,2] := 2.0;
   DATA[324,3] := 2.0;
   DATA[324,4] := 262.0482;
   DATA[324,5] := 8.393553;
   DATA[324,6] := 328.1723;
   DATA[324,7] := 2.440137;
   DATA[324,8] := 2.0;
   DATA[324,9] := 2.0;
   DATA[324,10] := 2.0;
   DATA[324,11] := 19.70037;
   DATA[324,12] := 2.209269;
   DATA[324,13] := 971.5458;
   DATA[324,14] := 1.0;
   DATA[324,15] := 2.0;
   DATA[324,16] := 1.0;
   DATA[324,17] := 1.0;
   DATA[324,18] := 1.0;
   DATA[324,19] := 2.0;
   DATA[324,20] := 148.808;
   DATA[324,21] := 155.8575;
   DATA[324,22] := 1.714158;
   DATA[324,23] := 970.4819;
   DATA[324,24] := 2.0;
   DATA[324,25] := 2.0;
   DATA[324,26] := 7.878942;
   DATA[324,27] := 145.1679;
   DATA[324,28] := 263.7465;
   DATA[324,29] := 12.03538;
   DATA[324,30] := 1.728275;
   DATA[324,31] := 1.271423;
   DATA[324,32] := 0.7352687;
   DATA[324,33] := 0.3080421;
   DATA[324,34] := 2.0;
   DATA[324,35] := 250.9132;
   DATA[324,36] := 1.69801;
   DATA[324,37] := 189.5988;
   DATA[324,38] := 0.000128152;
   DATA[324,39] := 1.0;
   DATA[325,0] := 2.585914;
   DATA[325,1] := 527.3608;
   DATA[325,2] := 2.0;
   DATA[325,3] := 2.0;
   DATA[325,4] := 262.0482;
   DATA[325,5] := 8.390669;
   DATA[325,6] := 328.1723;
   DATA[325,7] := 2.440137;
   DATA[325,8] := 2.0;
   DATA[325,9] := 2.0;
   DATA[325,10] := 2.0;
   DATA[325,11] := 19.70037;
   DATA[325,12] := 2.209525;
   DATA[325,13] := 971.746;
   DATA[325,14] := 1.0;
   DATA[325,15] := 2.0;
   DATA[325,16] := 1.0;
   DATA[325,17] := 1.0;
   DATA[325,18] := 1.0;
   DATA[325,19] := 2.0;
   DATA[325,20] := 148.808;
   DATA[325,21] := 155.9344;
   DATA[325,22] := 1.714158;
   DATA[325,23] := 970.5973;
   DATA[325,24] := 2.0;
   DATA[325,25] := 2.0;
   DATA[325,26] := 7.878942;
   DATA[325,27] := 144.9628;
   DATA[325,28] := 263.7465;
   DATA[325,29] := 12.03538;
   DATA[325,30] := 1.728275;
   DATA[325,31] := 1.271423;
   DATA[325,32] := 0.7352687;
   DATA[325,33] := 0.3084265;
   DATA[325,34] := 2.0;
   DATA[325,35] := 250.9132;
   DATA[325,36] := 1.69801;
   DATA[325,37] := 189.5988;
   DATA[325,38] := 0.000128152;
   DATA[325,39] := 1.0;
   DATA[326,0] := 2.566377;
   DATA[326,1] := 527.7926;
   DATA[326,2] := 2.0;
   DATA[326,3] := 2.0;
   DATA[326,4] := 262.0482;
   DATA[326,5] := 8.390669;
   DATA[326,6] := 328.1723;
   DATA[326,7] := 2.440137;
   DATA[326,8] := 2.0;
   DATA[326,9] := 2.0;
   DATA[326,10] := 2.0;
   DATA[326,11] := 19.70037;
   DATA[326,12] := 2.210678;
   DATA[326,13] := 971.8262;
   DATA[326,14] := 1.0;
   DATA[326,15] := 2.0;
   DATA[326,16] := 1.0;
   DATA[326,17] := 1.0;
   DATA[326,18] := 1.0;
   DATA[326,19] := 2.0;
   DATA[326,20] := 148.808;
   DATA[326,21] := 155.9344;
   DATA[326,22] := 1.714158;
   DATA[326,23] := 970.9434;
   DATA[326,24] := 2.0;
   DATA[326,25] := 2.0;
   DATA[326,26] := 7.878942;
   DATA[326,27] := 144.9116;
   DATA[326,28] := 263.7465;
   DATA[326,29] := 12.03538;
   DATA[326,30] := 1.728275;
   DATA[326,31] := 1.271423;
   DATA[326,32] := 0.7352687;
   DATA[326,33] := 0.3084265;
   DATA[326,34] := 2.0;
   DATA[326,35] := 250.9132;
   DATA[326,36] := 1.69801;
   DATA[326,37] := 189.5988;
   DATA[326,38] := 0.000128152;
   DATA[326,39] := 1.0;
   DATA[327,0] := 2.553886;
   DATA[327,1] := 528.1851;
   DATA[327,2] := 2.0;
   DATA[327,3] := 2.0;
   DATA[327,4] := 262.0482;
   DATA[327,5] := 8.390669;
   DATA[327,6] := 328.1723;
   DATA[327,7] := 2.440137;
   DATA[327,8] := 2.0;
   DATA[327,9] := 2.0;
   DATA[327,10] := 2.0;
   DATA[327,11] := 19.70037;
   DATA[327,12] := 2.210678;
   DATA[327,13] := 971.8662;
   DATA[327,14] := 1.0;
   DATA[327,15] := 2.0;
   DATA[327,16] := 1.0;
   DATA[327,17] := 1.0;
   DATA[327,18] := 1.0;
   DATA[327,19] := 2.0;
   DATA[327,20] := 148.808;
   DATA[327,21] := 155.9344;
   DATA[327,22] := 1.714158;
   DATA[327,23] := 971.0972;
   DATA[327,24] := 2.0;
   DATA[327,25] := 2.0;
   DATA[327,26] := 7.878942;
   DATA[327,27] := 144.9116;
   DATA[327,28] := 263.7465;
   DATA[327,29] := 12.03538;
   DATA[327,30] := 1.729172;
   DATA[327,31] := 1.271423;
   DATA[327,32] := 0.7352687;
   DATA[327,33] := 0.3084265;
   DATA[327,34] := 2.0;
   DATA[327,35] := 250.9132;
   DATA[327,36] := 1.69801;
   DATA[327,37] := 189.6469;
   DATA[327,38] := 0.000128152;
   DATA[327,39] := 1.0;
   DATA[328,0] := 2.536271;
   DATA[328,1] := 528.6169;
   DATA[328,2] := 2.0;
   DATA[328,3] := 2.0;
   DATA[328,4] := 262.0482;
   DATA[328,5] := 8.390669;
   DATA[328,6] := 328.1723;
   DATA[328,7] := 2.440137;
   DATA[328,8] := 2.0;
   DATA[328,9] := 2.0;
   DATA[328,10] := 2.0;
   DATA[328,11] := 19.77079;
   DATA[328,12] := 2.210678;
   DATA[328,13] := 971.8262;
   DATA[328,14] := 1.0;
   DATA[328,15] := 2.0;
   DATA[328,16] := 1.0;
   DATA[328,17] := 1.0;
   DATA[328,18] := 1.0;
   DATA[328,19] := 2.0;
   DATA[328,20] := 148.808;
   DATA[328,21] := 155.9344;
   DATA[328,22] := 1.714158;
   DATA[328,23] := 970.9818;
   DATA[328,24] := 2.0;
   DATA[328,25] := 2.0;
   DATA[328,26] := 7.878942;
   DATA[328,27] := 144.9116;
   DATA[328,28] := 263.7465;
   DATA[328,29] := 12.03538;
   DATA[328,30] := 1.729172;
   DATA[328,31] := 1.264378;
   DATA[328,32] := 0.7352687;
   DATA[328,33] := 0.3066329;
   DATA[328,34] := 2.0;
   DATA[328,35] := 250.9132;
   DATA[328,36] := 1.69801;
   DATA[328,37] := 189.8071;
   DATA[328,38] := 0.000128152;
   DATA[328,39] := 1.0;
   DATA[329,0] := 2.518015;
   DATA[329,1] := 529.0486;
   DATA[329,2] := 2.0;
   DATA[329,3] := 2.0;
   DATA[329,4] := 262.0482;
   DATA[329,5] := 8.391951;
   DATA[329,6] := 328.1723;
   DATA[329,7] := 2.440137;
   DATA[329,8] := 2.0;
   DATA[329,9] := 2.0;
   DATA[329,10] := 2.0;
   DATA[329,11] := 19.77079;
   DATA[329,12] := 2.210678;
   DATA[329,13] := 971.6259;
   DATA[329,14] := 1.0;
   DATA[329,15] := 2.0;
   DATA[329,16] := 1.0;
   DATA[329,17] := 1.0;
   DATA[329,18] := 1.0;
   DATA[329,19] := 2.0;
   DATA[329,20] := 148.808;
   DATA[329,21] := 155.8318;
   DATA[329,22] := 1.714158;
   DATA[329,23] := 970.7511;
   DATA[329,24] := 2.0;
   DATA[329,25] := 2.0;
   DATA[329,26] := 7.878942;
   DATA[329,27] := 144.9116;
   DATA[329,28] := 263.7465;
   DATA[329,29] := 12.03538;
   DATA[329,30] := 1.729172;
   DATA[329,31] := 1.254515;
   DATA[329,32] := 0.7352687;
   DATA[329,33] := 0.3066329;
   DATA[329,34] := 2.0;
   DATA[329,35] := 251.0574;
   DATA[329,36] := 1.69801;
   DATA[329,37] := 189.8071;
   DATA[329,38] := 0.000128152;
   DATA[329,39] := 1.0;
   DATA[330,0] := 2.494635;
   DATA[330,1] := 529.559;
   DATA[330,2] := 2.0;
   DATA[330,3] := 2.0;
   DATA[330,4] := 262.0482;
   DATA[330,5] := 8.393553;
   DATA[330,6] := 328.1723;
   DATA[330,7] := 2.442316;
   DATA[330,8] := 2.0;
   DATA[330,9] := 2.0;
   DATA[330,10] := 2.0;
   DATA[330,11] := 19.77079;
   DATA[330,12] := 2.210678;
   DATA[330,13] := 971.4256;
   DATA[330,14] := 1.0;
   DATA[330,15] := 2.0;
   DATA[330,16] := 1.0;
   DATA[330,17] := 1.0;
   DATA[330,18] := 1.0;
   DATA[330,19] := 2.0;
   DATA[330,20] := 148.808;
   DATA[330,21] := 155.8318;
   DATA[330,22] := 1.717105;
   DATA[330,23] := 970.7511;
   DATA[330,24] := 2.0;
   DATA[330,25] := 2.0;
   DATA[330,26] := 7.878942;
   DATA[330,27] := 144.9628;
   DATA[330,28] := 263.7465;
   DATA[330,29] := 12.03538;
   DATA[330,30] := 1.729172;
   DATA[330,31] := 1.254003;
   DATA[330,32] := 0.7352687;
   DATA[330,33] := 0.3066329;
   DATA[330,34] := 2.0;
   DATA[330,35] := 251.0574;
   DATA[330,36] := 1.69801;
   DATA[330,37] := 189.8071;
   DATA[330,38] := 0.000128152;
   DATA[330,39] := 1.0;
   DATA[331,0] := 2.483105;
   DATA[331,1] := 530.1085;
   DATA[331,2] := 2.0;
   DATA[331,3] := 2.0;
   DATA[331,4] := 262.0482;
   DATA[331,5] := 8.393553;
   DATA[331,6] := 328.1723;
   DATA[331,7] := 2.442956;
   DATA[331,8] := 2.0;
   DATA[331,9] := 2.0;
   DATA[331,10] := 2.0;
   DATA[331,11] := 19.77079;
   DATA[331,12] := 2.210678;
   DATA[331,13] := 971.1453;
   DATA[331,14] := 1.0;
   DATA[331,15] := 2.0;
   DATA[331,16] := 1.0;
   DATA[331,17] := 1.0;
   DATA[331,18] := 1.0;
   DATA[331,19] := 2.0;
   DATA[331,20] := 148.808;
   DATA[331,21] := 155.8318;
   DATA[331,22] := 1.718387;
   DATA[331,23] := 970.9434;
   DATA[331,24] := 2.0;
   DATA[331,25] := 2.0;
   DATA[331,26] := 7.878942;
   DATA[331,27] := 145.1679;
   DATA[331,28] := 263.7465;
   DATA[331,29] := 12.03538;
   DATA[331,30] := 1.729172;
   DATA[331,31] := 1.253619;
   DATA[331,32] := 0.7352687;
   DATA[331,33] := 0.3066329;
   DATA[331,34] := 2.0;
   DATA[331,35] := 251.0574;
   DATA[331,36] := 1.69801;
   DATA[331,37] := 189.8071;
   DATA[331,38] := 0.000128152;
   DATA[331,39] := 1.0;
   DATA[332,0] := 2.464209;
   DATA[332,1] := 530.7758;
   DATA[332,2] := 2.0;
   DATA[332,3] := 2.0;
   DATA[332,4] := 262.0482;
   DATA[332,5] := 8.393553;
   DATA[332,6] := 328.1723;
   DATA[332,7] := 2.442956;
   DATA[332,8] := 2.0;
   DATA[332,9] := 2.0;
   DATA[332,10] := 2.0;
   DATA[332,11] := 19.77079;
   DATA[332,12] := 2.210678;
   DATA[332,13] := 971.1853;
   DATA[332,14] := 1.0;
   DATA[332,15] := 2.0;
   DATA[332,16] := 1.0;
   DATA[332,17] := 1.0;
   DATA[332,18] := 1.0;
   DATA[332,19] := 2.0;
   DATA[332,20] := 148.808;
   DATA[332,21] := 155.8318;
   DATA[332,22] := 1.718387;
   DATA[332,23] := 970.8665;
   DATA[332,24] := 2.0;
   DATA[332,25] := 2.0;
   DATA[332,26] := 7.878942;
   DATA[332,27] := 145.1679;
   DATA[332,28] := 263.7465;
   DATA[332,29] := 12.03538;
   DATA[332,30] := 1.729172;
   DATA[332,31] := 1.260664;
   DATA[332,32] := 0.7352687;
   DATA[332,33] := 0.3066329;
   DATA[332,34] := 2.0;
   DATA[332,35] := 251.0574;
   DATA[332,36] := 1.826162;
   DATA[332,37] := 189.8071;
   DATA[332,38] := 0.000128152;
   DATA[332,39] := 1.0;
   DATA[333,0] := 2.45428;
   DATA[333,1] := 530.9328;
   DATA[333,2] := 2.0;
   DATA[333,3] := 2.0;
   DATA[333,4] := 262.0482;
   DATA[333,5] := 8.393553;
   DATA[333,6] := 328.1723;
   DATA[333,7] := 2.442956;
   DATA[333,8] := 2.0;
   DATA[333,9] := 2.0;
   DATA[333,10] := 2.0;
   DATA[333,11] := 19.66835;
   DATA[333,12] := 2.210678;
   DATA[333,13] := 971.3856;
   DATA[333,14] := 1.0;
   DATA[333,15] := 2.0;
   DATA[333,16] := 1.0;
   DATA[333,17] := 1.0;
   DATA[333,18] := 1.0;
   DATA[333,19] := 2.0;
   DATA[333,20] := 148.808;
   DATA[333,21] := 155.8318;
   DATA[333,22] := 1.718387;
   DATA[333,23] := 970.7126;
   DATA[333,24] := 2.0;
   DATA[333,25] := 2.0;
   DATA[333,26] := 7.880864;
   DATA[333,27] := 145.1679;
   DATA[333,28] := 263.7465;
   DATA[333,29] := 12.03538;
   DATA[333,30] := 1.729172;
   DATA[333,31] := 1.28167;
   DATA[333,32] := 0.7352687;
   DATA[333,33] := 0.3066329;
   DATA[333,34] := 2.0;
   DATA[333,35] := 251.0574;
   DATA[333,36] := 1.826162;
   DATA[333,37] := 189.8071;
   DATA[333,38] := 0.000128152;
   DATA[333,39] := 1.0;
   DATA[334,0] := 2.435064;
   DATA[334,1] := 531.3253;
   DATA[334,2] := 2.0;
   DATA[334,3] := 2.0;
   DATA[334,4] := 262.0482;
   DATA[334,5] := 8.393553;
   DATA[334,6] := 328.1723;
   DATA[334,7] := 2.441803;
   DATA[334,8] := 2.0;
   DATA[334,9] := 2.0;
   DATA[334,10] := 2.0;
   DATA[334,11] := 19.62674;
   DATA[334,12] := 2.210166;
   DATA[334,13] := 970.985;
   DATA[334,14] := 1.0;
   DATA[334,15] := 2.0;
   DATA[334,16] := 1.0;
   DATA[334,17] := 1.0;
   DATA[334,18] := 1.0;
   DATA[334,19] := 2.0;
   DATA[334,20] := 148.808;
   DATA[334,21] := 155.8575;
   DATA[334,22] := 1.718387;
   DATA[334,23] := 970.405;
   DATA[334,24] := 2.0;
   DATA[334,25] := 2.0;
   DATA[334,26] := 7.880864;
   DATA[334,27] := 145.0397;
   DATA[334,28] := 263.7465;
   DATA[334,29] := 12.03538;
   DATA[334,30] := 1.729172;
   DATA[334,31] := 1.300243;
   DATA[334,32] := 0.7352687;
   DATA[334,33] := 0.3066329;
   DATA[334,34] := 2.0;
   DATA[334,35] := 251.0574;
   DATA[334,36] := 1.826162;
   DATA[334,37] := 189.7751;
   DATA[334,38] := 0.000128152;
   DATA[334,39] := 1.0;
   DATA[335,0] := 2.424174;
   DATA[335,1] := 531.8749;
   DATA[335,2] := 2.0;
   DATA[335,3] := 2.0;
   DATA[335,4] := 262.0482;
   DATA[335,5] := 8.393553;
   DATA[335,6] := 328.1723;
   DATA[335,7] := 2.441803;
   DATA[335,8] := 2.0;
   DATA[335,9] := 2.0;
   DATA[335,10] := 2.0;
   DATA[335,11] := 19.56271;
   DATA[335,12] := 2.210166;
   DATA[335,13] := 970.9449;
   DATA[335,14] := 1.0;
   DATA[335,15] := 2.0;
   DATA[335,16] := 1.0;
   DATA[335,17] := 1.0;
   DATA[335,18] := 1.0;
   DATA[335,19] := 2.0;
   DATA[335,20] := 148.808;
   DATA[335,21] := 155.8575;
   DATA[335,22] := 1.718387;
   DATA[335,23] := 970.2897;
   DATA[335,24] := 2.0;
   DATA[335,25] := 2.0;
   DATA[335,26] := 7.880864;
   DATA[335,27] := 145.0397;
   DATA[335,28] := 263.7465;
   DATA[335,29] := 12.03538;
   DATA[335,30] := 1.729172;
   DATA[335,31] := 1.318945;
   DATA[335,32] := 0.7352687;
   DATA[335,33] := 0.3081062;
   DATA[335,34] := 2.0;
   DATA[335,35] := 251.0574;
   DATA[335,36] := 1.762086;
   DATA[335,37] := 189.759;
   DATA[335,38] := 0.000128152;
   DATA[335,39] := 1.0;
   DATA[336,0] := 2.422253;
   DATA[336,1] := 532.1497;
   DATA[336,2] := 2.0;
   DATA[336,3] := 2.0;
   DATA[336,4] := 262.0482;
   DATA[336,5] := 8.393553;
   DATA[336,6] := 328.1723;
   DATA[336,7] := 2.440393;
   DATA[336,8] := 2.0;
   DATA[336,9] := 2.0;
   DATA[336,10] := 2.0;
   DATA[336,11] := 19.56271;
   DATA[336,12] := 2.209525;
   DATA[336,13] := 970.5444;
   DATA[336,14] := 1.0;
   DATA[336,15] := 2.0;
   DATA[336,16] := 1.0;
   DATA[336,17] := 1.0;
   DATA[336,18] := 1.0;
   DATA[336,19] := 2.0;
   DATA[336,20] := 148.808;
   DATA[336,21] := 156.0625;
   DATA[336,22] := 1.717874;
   DATA[336,23] := 969.9052;
   DATA[336,24] := 2.0;
   DATA[336,25] := 2.0;
   DATA[336,26] := 7.880864;
   DATA[336,27] := 145.0397;
   DATA[336,28] := 263.7465;
   DATA[336,29] := 12.03538;
   DATA[336,30] := 1.729172;
   DATA[336,31] := 1.315742;
   DATA[336,32] := 0.7352687;
   DATA[336,33] := 0.3084905;
   DATA[336,34] := 2.0;
   DATA[336,35] := 251.0574;
   DATA[336,36] := 1.69801;
   DATA[336,37] := 189.759;
   DATA[336,38] := 0.000128152;
   DATA[336,39] := 1.0;
   DATA[337,0] := 2.422253;
   DATA[337,1] := 532.3851;
   DATA[337,2] := 2.0;
   DATA[337,3] := 2.0;
   DATA[337,4] := 262.0482;
   DATA[337,5] := 8.394835;
   DATA[337,6] := 328.1723;
   DATA[337,7] := 2.440393;
   DATA[337,8] := 2.0;
   DATA[337,9] := 2.0;
   DATA[337,10] := 2.0;
   DATA[337,11] := 19.57232;
   DATA[337,12] := 2.207475;
   DATA[337,13] := 970.3842;
   DATA[337,14] := 1.0;
   DATA[337,15] := 2.0;
   DATA[337,16] := 1.0;
   DATA[337,17] := 1.0;
   DATA[337,18] := 1.0;
   DATA[337,19] := 2.0;
   DATA[337,20] := 148.808;
   DATA[337,21] := 156.0625;
   DATA[337,22] := 1.716721;
   DATA[337,23] := 969.4437;
   DATA[337,24] := 2.0;
   DATA[337,25] := 2.0;
   DATA[337,26] := 7.880864;
   DATA[337,27] := 145.0397;
   DATA[337,28] := 263.7465;
   DATA[337,29] := 12.03538;
   DATA[337,30] := 1.729172;
   DATA[337,31] := 1.29512;
   DATA[337,32] := 0.7352687;
   DATA[337,33] := 0.3070813;
   DATA[337,34] := 2.0;
   DATA[337,35] := 251.0574;
   DATA[337,36] := 1.69801;
   DATA[337,37] := 189.759;
   DATA[337,38] := 0.000128152;
   DATA[337,39] := 1.0;
   DATA[338,0] := 2.456202;
   DATA[338,1] := 532.5029;
   DATA[338,2] := 2.0;
   DATA[338,3] := 2.0;
   DATA[338,4] := 262.0482;
   DATA[338,5] := 8.394835;
   DATA[338,6] := 328.1723;
   DATA[338,7] := 2.440393;
   DATA[338,8] := 2.0;
   DATA[338,9] := 2.0;
   DATA[338,10] := 2.0;
   DATA[338,11] := 19.59472;
   DATA[338,12] := 2.206322;
   DATA[338,13] := 970.8649;
   DATA[338,14] := 1.0;
   DATA[338,15] := 2.0;
   DATA[338,16] := 1.0;
   DATA[338,17] := 1.0;
   DATA[338,18] := 1.0;
   DATA[338,19] := 2.0;
   DATA[338,20] := 148.808;
   DATA[338,21] := 156.0625;
   DATA[338,22] := 1.715824;
   DATA[338,23] := 969.5206;
   DATA[338,24] := 2.0;
   DATA[338,25] := 2.0;
   DATA[338,26] := 7.880864;
   DATA[338,27] := 145.0397;
   DATA[338,28] := 263.7465;
   DATA[338,29] := 12.03538;
   DATA[338,30] := 1.729172;
   DATA[338,31] := 1.296657;
   DATA[338,32] := 0.7352687;
   DATA[338,33] := 0.3070813;
   DATA[338,34] := 2.0;
   DATA[338,35] := 251.0574;
   DATA[338,36] := 1.69801;
   DATA[338,37] := 189.759;
   DATA[338,38] := 0.000128152;
   DATA[338,39] := 1.0;
   DATA[339,0] := 2.505204;
   DATA[339,1] := 532.4637;
   DATA[339,2] := 2.0;
   DATA[339,3] := 2.0;
   DATA[339,4] := 262.0482;
   DATA[339,5] := 8.394835;
   DATA[339,6] := 328.1723;
   DATA[339,7] := 2.440137;
   DATA[339,8] := 2.0;
   DATA[339,9] := 2.0;
   DATA[339,10] := 2.0;
   DATA[339,11] := 19.59472;
   DATA[339,12] := 2.206322;
   DATA[339,13] := 970.5444;
   DATA[339,14] := 1.0;
   DATA[339,15] := 2.0;
   DATA[339,16] := 1.0;
   DATA[339,17] := 1.0;
   DATA[339,18] := 1.0;
   DATA[339,19] := 2.0;
   DATA[339,20] := 148.808;
   DATA[339,21] := 155.7806;
   DATA[339,22] := 1.715824;
   DATA[339,23] := 969.4053;
   DATA[339,24] := 2.0;
   DATA[339,25] := 2.0;
   DATA[339,26] := 7.880864;
   DATA[339,27] := 145.0397;
   DATA[339,28] := 263.7465;
   DATA[339,29] := 12.03538;
   DATA[339,30] := 1.729172;
   DATA[339,31] := 1.29512;
   DATA[339,32] := 0.7352687;
   DATA[339,33] := 0.3070813;
   DATA[339,34] := 2.0;
   DATA[339,35] := 251.0574;
   DATA[339,36] := 1.69801;
   DATA[339,37] := 189.759;
   DATA[339,38] := 0.000128152;
   DATA[339,39] := 1.0;
   DATA[340,0] := 2.54652;
   DATA[340,1] := 532.6992;
   DATA[340,2] := 2.0;
   DATA[340,3] := 2.0;
   DATA[340,4] := 262.0482;
   DATA[340,5] := 8.394835;
   DATA[340,6] := 328.1723;
   DATA[340,7] := 2.439112;
   DATA[340,8] := 2.0;
   DATA[340,9] := 2.0;
   DATA[340,10] := 2.0;
   DATA[340,11] := 19.59472;
   DATA[340,12] := 2.208628;
   DATA[340,13] := 970.5444;
   DATA[340,14] := 1.0;
   DATA[340,15] := 2.0;
   DATA[340,16] := 1.0;
   DATA[340,17] := 1.0;
   DATA[340,18] := 1.0;
   DATA[340,19] := 2.0;
   DATA[340,20] := 148.808;
   DATA[340,21] := 155.7806;
   DATA[340,22] := 1.715824;
   DATA[340,23] := 969.4053;
   DATA[340,24] := 2.0;
   DATA[340,25] := 2.0;
   DATA[340,26] := 7.880864;
   DATA[340,27] := 145.0397;
   DATA[340,28] := 263.7465;
   DATA[340,29] := 12.03538;
   DATA[340,30] := 1.729172;
   DATA[340,31] := 1.298962;
   DATA[340,32] := 0.7352687;
   DATA[340,33] := 0.3070813;
   DATA[340,34] := 2.0;
   DATA[340,35] := 251.0574;
   DATA[340,36] := 1.746067;
   DATA[340,37] := 189.759;
   DATA[340,38] := 0.000128152;
   DATA[340,39] := 1.0;
   DATA[341,0] := 2.577907;
   DATA[341,1] := 532.2674;
   DATA[341,2] := 2.0;
   DATA[341,3] := 2.0;
   DATA[341,4] := 262.0482;
   DATA[341,5] := 8.394835;
   DATA[341,6] := 328.1723;
   DATA[341,7] := 2.439112;
   DATA[341,8] := 2.0;
   DATA[341,9] := 2.0;
   DATA[341,10] := 2.0;
   DATA[341,11] := 19.60753;
   DATA[341,12] := 2.209013;
   DATA[341,13] := 970.7447;
   DATA[341,14] := 1.0;
   DATA[341,15] := 2.0;
   DATA[341,16] := 1.0;
   DATA[341,17] := 1.0;
   DATA[341,18] := 1.0;
   DATA[341,19] := 2.0;
   DATA[341,20] := 148.808;
   DATA[341,21] := 155.7806;
   DATA[341,22] := 1.715824;
   DATA[341,23] := 969.4437;
   DATA[341,24] := 2.0;
   DATA[341,25] := 2.0;
   DATA[341,26] := 7.880864;
   DATA[341,27] := 145.0397;
   DATA[341,28] := 263.7465;
   DATA[341,29] := 12.03538;
   DATA[341,30] := 1.729172;
   DATA[341,31] := 1.302037;
   DATA[341,32] := 0.7352687;
   DATA[341,33] := 0.3065048;
   DATA[341,34] := 2.0;
   DATA[341,35] := 251.0574;
   DATA[341,36] := 1.746067;
   DATA[341,37] := 189.6629;
   DATA[341,38] := 0.000128152;
   DATA[341,39] := 1.0;
   DATA[342,0] := 2.621785;
   DATA[342,1] := 531.9141;
   DATA[342,2] := 2.0;
   DATA[342,3] := 2.0;
   DATA[342,4] := 262.0482;
   DATA[342,5] := 8.394835;
   DATA[342,6] := 328.1723;
   DATA[342,7] := 2.439112;
   DATA[342,8] := 2.0;
   DATA[342,9] := 2.0;
   DATA[342,10] := 2.0;
   DATA[342,11] := 19.63954;
   DATA[342,12] := 2.209013;
   DATA[342,13] := 970.8248;
   DATA[342,14] := 1.0;
   DATA[342,15] := 2.0;
   DATA[342,16] := 1.0;
   DATA[342,17] := 1.0;
   DATA[342,18] := 1.0;
   DATA[342,19] := 2.0;
   DATA[342,20] := 148.808;
   DATA[342,21] := 155.7806;
   DATA[342,22] := 1.716592;
   DATA[342,23] := 969.5591;
   DATA[342,24] := 2.0;
   DATA[342,25] := 2.0;
   DATA[342,26] := 7.880864;
   DATA[342,27] := 145.0397;
   DATA[342,28] := 263.7465;
   DATA[342,29] := 12.03538;
   DATA[342,30] := 1.729172;
   DATA[342,31] := 1.311003;
   DATA[342,32] := 0.7352687;
   DATA[342,33] := 0.3065048;
   DATA[342,34] := 2.0;
   DATA[342,35] := 250.9773;
   DATA[342,36] := 1.746067;
   DATA[342,37] := 189.6629;
   DATA[342,38] := 0.000128152;
   DATA[342,39] := 1.0;
   DATA[343,0] := 2.651251;
   DATA[343,1] := 531.7571;
   DATA[343,2] := 2.0;
   DATA[343,3] := 2.0;
   DATA[343,4] := 262.0482;
   DATA[343,5] := 8.394835;
   DATA[343,6] := 328.1723;
   DATA[343,7] := 2.43924;
   DATA[343,8] := 2.0;
   DATA[343,9] := 2.0;
   DATA[343,10] := 2.0;
   DATA[343,11] := 19.65235;
   DATA[343,12] := 2.211959;
   DATA[343,13] := 970.985;
   DATA[343,14] := 1.0;
   DATA[343,15] := 2.0;
   DATA[343,16] := 1.0;
   DATA[343,17] := 1.0;
   DATA[343,18] := 1.0;
   DATA[343,19] := 2.0;
   DATA[343,20] := 148.808;
   DATA[343,21] := 155.8318;
   DATA[343,22] := 1.716592;
   DATA[343,23] := 969.4053;
   DATA[343,24] := 2.0;
   DATA[343,25] := 2.0;
   DATA[343,26] := 7.880864;
   DATA[343,27] := 145.0397;
   DATA[343,28] := 263.7465;
   DATA[343,29] := 12.15073;
   DATA[343,30] := 1.729172;
   DATA[343,31] := 1.306776;
   DATA[343,32] := 0.7352687;
   DATA[343,33] := 0.3065048;
   DATA[343,34] := 2.0;
   DATA[343,35] := 250.9773;
   DATA[343,36] := 1.746067;
   DATA[343,37] := 189.6629;
   DATA[343,38] := 0.000128152;
   DATA[343,39] := 1.0;
   DATA[344,0] := 2.670788;
   DATA[344,1] := 531.4824;
   DATA[344,2] := 2.0;
   DATA[344,3] := 2.0;
   DATA[344,4] := 262.0482;
   DATA[344,5] := 8.394835;
   DATA[344,6] := 328.1723;
   DATA[344,7] := 2.439753;
   DATA[344,8] := 2.0;
   DATA[344,9] := 2.0;
   DATA[344,10] := 2.0;
   DATA[344,11] := 19.65235;
   DATA[344,12] := 2.212856;
   DATA[344,13] := 971.1453;
   DATA[344,14] := 1.0;
   DATA[344,15] := 2.0;
   DATA[344,16] := 1.0;
   DATA[344,17] := 1.0;
   DATA[344,18] := 1.0;
   DATA[344,19] := 2.0;
   DATA[344,20] := 148.808;
   DATA[344,21] := 155.9087;
   DATA[344,22] := 1.716592;
   DATA[344,23] := 969.7898;
   DATA[344,24] := 2.0;
   DATA[344,25] := 2.0;
   DATA[344,26] := 7.880864;
   DATA[344,27] := 145.0397;
   DATA[344,28] := 263.7465;
   DATA[344,29] := 12.15073;
   DATA[344,30] := 1.729172;
   DATA[344,31] := 1.301396;
   DATA[344,32] := 0.7352687;
   DATA[344,33] := 0.3065048;
   DATA[344,34] := 2.0;
   DATA[344,35] := 250.9773;
   DATA[344,36] := 1.746067;
   DATA[344,37] := 189.6629;
   DATA[344,38] := 0.000128152;
   DATA[344,39] := 1.0;
   DATA[345,0] := 2.670788;
   DATA[345,1] := 531.0113;
   DATA[345,2] := 2.0;
   DATA[345,3] := 2.0;
   DATA[345,4] := 262.0482;
   DATA[345,5] := 8.393553;
   DATA[345,6] := 328.1723;
   DATA[345,7] := 2.441419;
   DATA[345,8] := 2.0;
   DATA[345,9] := 2.0;
   DATA[345,10] := 2.0;
   DATA[345,11] := 19.67155;
   DATA[345,12] := 2.212856;
   DATA[345,13] := 971.7861;
   DATA[345,14] := 1.0;
   DATA[345,15] := 2.0;
   DATA[345,16] := 1.0;
   DATA[345,17] := 1.0;
   DATA[345,18] := 1.0;
   DATA[345,19] := 2.0;
   DATA[345,20] := 148.808;
   DATA[345,21] := 155.9087;
   DATA[345,22] := 1.716592;
   DATA[345,23] := 969.7513;
   DATA[345,24] := 2.0;
   DATA[345,25] := 2.0;
   DATA[345,26] := 7.880864;
   DATA[345,27] := 145.0397;
   DATA[345,28] := 263.7465;
   DATA[345,29] := 12.15073;
   DATA[345,30] := 1.728916;
   DATA[345,31] := 1.292558;
   DATA[345,32] := 0.7352687;
   DATA[345,33] := 0.3065048;
   DATA[345,34] := 2.0;
   DATA[345,35] := 250.9453;
   DATA[345,36] := 1.746067;
   DATA[345,37] := 189.6629;
   DATA[345,38] := 0.000128152;
   DATA[345,39] := 1.0;
   DATA[346,0] := 2.645165;
   DATA[346,1] := 530.9328;
   DATA[346,2] := 2.0;
   DATA[346,3] := 2.0;
   DATA[346,4] := 262.0482;
   DATA[346,5] := 8.393232;
   DATA[346,6] := 328.1723;
   DATA[346,7] := 2.441419;
   DATA[346,8] := 2.0;
   DATA[346,9] := 2.0;
   DATA[346,10] := 2.0;
   DATA[346,11] := 19.67796;
   DATA[346,12] := 2.212856;
   DATA[346,13] := 971.666;
   DATA[346,14] := 1.0;
   DATA[346,15] := 2.0;
   DATA[346,16] := 1.0;
   DATA[346,17] := 1.0;
   DATA[346,18] := 1.0;
   DATA[346,19] := 2.0;
   DATA[346,20] := 148.808;
   DATA[346,21] := 155.9087;
   DATA[346,22] := 1.716592;
   DATA[346,23] := 969.5206;
   DATA[346,24] := 2.0;
   DATA[346,25] := 2.0;
   DATA[346,26] := 7.879582;
   DATA[346,27] := 145.0397;
   DATA[346,28] := 263.7465;
   DATA[346,29] := 12.15073;
   DATA[346,30] := 1.726865;
   DATA[346,31] := 1.281798;
   DATA[346,32] := 0.7366771;
   DATA[346,33] := 0.306761;
   DATA[346,34] := 2.0;
   DATA[346,35] := 250.8972;
   DATA[346,36] := 1.746067;
   DATA[346,37] := 189.6629;
   DATA[346,38] := 0.000128152;
   DATA[346,39] := 1.0;
   DATA[347,0] := 2.632995;
   DATA[347,1] := 530.344;
   DATA[347,2] := 2.0;
   DATA[347,3] := 2.0;
   DATA[347,4] := 262.0482;
   DATA[347,5] := 8.393232;
   DATA[347,6] := 328.1723;
   DATA[347,7] := 2.441419;
   DATA[347,8] := 2.0;
   DATA[347,9] := 2.0;
   DATA[347,10] := 2.0;
   DATA[347,11] := 19.70037;
   DATA[347,12] := 2.212856;
   DATA[347,13] := 971.9463;
   DATA[347,14] := 1.0;
   DATA[347,15] := 2.0;
   DATA[347,16] := 1.0;
   DATA[347,17] := 1.0;
   DATA[347,18] := 1.0;
   DATA[347,19] := 2.0;
   DATA[347,20] := 148.808;
   DATA[347,21] := 155.96;
   DATA[347,22] := 1.714542;
   DATA[347,23] := 969.4437;
   DATA[347,24] := 2.0;
   DATA[347,25] := 2.0;
   DATA[347,26] := 7.879582;
   DATA[347,27] := 145.0397;
   DATA[347,28] := 263.7465;
   DATA[347,29] := 12.15073;
   DATA[347,30] := 1.728147;
   DATA[347,31] := 1.286794;
   DATA[347,32] := 0.7379573;
   DATA[347,33] := 0.306761;
   DATA[347,34] := 2.0;
   DATA[347,35] := 250.8972;
   DATA[347,36] := 1.746067;
   DATA[347,37] := 189.6629;
   DATA[347,38] := 0.000128152;
   DATA[347,39] := 1.0;
   DATA[348,0] := 2.626589;
   DATA[348,1] := 529.8337;
   DATA[348,2] := 2.0;
   DATA[348,3] := 2.0;
   DATA[348,4] := 262.0482;
   DATA[348,5] := 8.393232;
   DATA[348,6] := 328.1723;
   DATA[348,7] := 2.441419;
   DATA[348,8] := 2.0;
   DATA[348,9] := 2.0;
   DATA[348,10] := 2.0;
   DATA[348,11] := 19.71637;
   DATA[348,12] := 2.212856;
   DATA[348,13] := 972.0264;
   DATA[348,14] := 1.0;
   DATA[348,15] := 2.0;
   DATA[348,16] := 1.0;
   DATA[348,17] := 1.0;
   DATA[348,18] := 1.0;
   DATA[348,19] := 2.0;
   DATA[348,20] := 148.808;
   DATA[348,21] := 155.96;
   DATA[348,22] := 1.714542;
   DATA[348,23] := 969.2515;
   DATA[348,24] := 2.0;
   DATA[348,25] := 2.0;
   DATA[348,26] := 7.879582;
   DATA[348,27] := 145.0397;
   DATA[348,28] := 263.7465;
   DATA[348,29] := 12.15073;
   DATA[348,30] := 1.728531;
   DATA[348,31] := 1.285641;
   DATA[348,32] := 0.7379573;
   DATA[348,33] := 0.306761;
   DATA[348,34] := 2.0;
   DATA[348,35] := 250.8972;
   DATA[348,36] := 1.746067;
   DATA[348,37] := 189.6629;
   DATA[348,38] := 0.000128152;
   DATA[348,39] := 1.0;
   DATA[349,0] := 2.626589;
   DATA[349,1] := 529.6375;
   DATA[349,2] := 2.0;
   DATA[349,3] := 2.0;
   DATA[349,4] := 262.0482;
   DATA[349,5] := 8.391951;
   DATA[349,6] := 328.3004;
   DATA[349,7] := 2.440521;
   DATA[349,8] := 2.0;
   DATA[349,9] := 2.0;
   DATA[349,10] := 2.0;
   DATA[349,11] := 19.71637;
   DATA[349,12] := 2.212856;
   DATA[349,13] := 971.8262;
   DATA[349,14] := 1.0;
   DATA[349,15] := 2.0;
   DATA[349,16] := 1.0;
   DATA[349,17] := 1.0;
   DATA[349,18] := 1.0;
   DATA[349,19] := 2.0;
   DATA[349,20] := 148.808;
   DATA[349,21] := 155.96;
   DATA[349,22] := 1.714542;
   DATA[349,23] := 969.5591;
   DATA[349,24] := 2.0;
   DATA[349,25] := 2.0;
   DATA[349,26] := 7.879582;
   DATA[349,27] := 145.0397;
   DATA[349,28] := 263.7465;
   DATA[349,29] := 12.15073;
   DATA[349,30] := 1.728531;
   DATA[349,31] := 1.281286;
   DATA[349,32] := 0.7379573;
   DATA[349,33] := 0.306761;
   DATA[349,34] := 2.0;
   DATA[349,35] := 250.8972;
   DATA[349,36] := 1.746067;
   DATA[349,37] := 189.5668;
   DATA[349,38] := 0.000128152;
   DATA[349,39] := 1.0;
   DATA[350,0] := 2.6157;
   DATA[350,1] := 529.3234;
   DATA[350,2] := 2.0;
   DATA[350,3] := 2.0;
   DATA[350,4] := 262.0482;
   DATA[350,5] := 8.391951;
   DATA[350,6] := 328.3004;
   DATA[350,7] := 2.440521;
   DATA[350,8] := 2.0;
   DATA[350,9] := 2.0;
   DATA[350,10] := 2.0;
   DATA[350,11] := 19.71637;
   DATA[350,12] := 2.212856;
   DATA[350,13] := 971.9463;
   DATA[350,14] := 1.0;
   DATA[350,15] := 2.0;
   DATA[350,16] := 1.0;
   DATA[350,17] := 1.0;
   DATA[350,18] := 1.0;
   DATA[350,19] := 2.0;
   DATA[350,20] := 148.808;
   DATA[350,21] := 155.96;
   DATA[350,22] := 1.714542;
   DATA[350,23] := 969.5975;
   DATA[350,24] := 2.0;
   DATA[350,25] := 2.0;
   DATA[350,26] := 7.879582;
   DATA[350,27] := 145.0397;
   DATA[350,28] := 263.7465;
   DATA[350,29] := 12.15073;
   DATA[350,30] := 1.725968;
   DATA[350,31] := 1.281286;
   DATA[350,32] := 0.7379573;
   DATA[350,33] := 0.306761;
   DATA[350,34] := 2.0;
   DATA[350,35] := 250.8972;
   DATA[350,36] := 1.746067;
   DATA[350,37] := 189.4867;
   DATA[350,38] := 0.000128152;
   DATA[350,39] := 1.0;
   DATA[351,0] := 2.592;
   DATA[351,1] := 529.4412;
   DATA[351,2] := 2.0;
   DATA[351,3] := 2.0;
   DATA[351,4] := 262.0482;
   DATA[351,5] := 8.391951;
   DATA[351,6] := 328.3004;
   DATA[351,7] := 2.440521;
   DATA[351,8] := 2.0;
   DATA[351,9] := 2.0;
   DATA[351,10] := 2.0;
   DATA[351,11] := 19.65235;
   DATA[351,12] := 2.209909;
   DATA[351,13] := 971.8662;
   DATA[351,14] := 1.0;
   DATA[351,15] := 2.0;
   DATA[351,16] := 1.0;
   DATA[351,17] := 1.0;
   DATA[351,18] := 1.0;
   DATA[351,19] := 2.0;
   DATA[351,20] := 148.808;
   DATA[351,21] := 155.96;
   DATA[351,22] := 1.714542;
   DATA[351,23] := 970.0205;
   DATA[351,24] := 2.0;
   DATA[351,25] := 2.0;
   DATA[351,26] := 7.879582;
   DATA[351,27] := 145.0397;
   DATA[351,28] := 263.7465;
   DATA[351,29] := 12.15073;
   DATA[351,30] := 1.725455;
   DATA[351,31] := 1.272064;
   DATA[351,32] := 0.7347566;
   DATA[351,33] := 0.3074656;
   DATA[351,34] := 2.0;
   DATA[351,35] := 250.8171;
   DATA[351,36] := 1.681991;
   DATA[351,37] := 189.4867;
   DATA[351,38] := 0.000128152;
   DATA[351,39] := 1.0;
   DATA[352,0] := 2.577907;
   DATA[352,1] := 529.2057;
   DATA[352,2] := 2.0;
   DATA[352,3] := 2.0;
   DATA[352,4] := 262.0482;
   DATA[352,5] := 8.391951;
   DATA[352,6] := 328.3004;
   DATA[352,7] := 2.439496;
   DATA[352,8] := 2.0;
   DATA[352,9] := 2.0;
   DATA[352,10] := 2.0;
   DATA[352,11] := 19.65235;
   DATA[352,12] := 2.209525;
   DATA[352,13] := 972.2267;
   DATA[352,14] := 1.0;
   DATA[352,15] := 2.0;
   DATA[352,16] := 1.0;
   DATA[352,17] := 1.0;
   DATA[352,18] := 1.0;
   DATA[352,19] := 2.0;
   DATA[352,20] := 148.808;
   DATA[352,21] := 155.96;
   DATA[352,22] := 1.716464;
   DATA[352,23] := 969.9052;
   DATA[352,24] := 2.0;
   DATA[352,25] := 2.0;
   DATA[352,26] := 7.879582;
   DATA[352,27] := 145.0397;
   DATA[352,28] := 263.7465;
   DATA[352,29] := 12.15073;
   DATA[352,30] := 1.724045;
   DATA[352,31] := 1.277059;
   DATA[352,32] := 0.7347566;
   DATA[352,33] := 0.3086186;
   DATA[352,34] := 2.0;
   DATA[352,35] := 250.785;
   DATA[352,36] := 1.617916;
   DATA[352,37] := 189.4546;
   DATA[352,38] := 0.000128152;
   DATA[352,39] := 1.0;
   DATA[353,0] := 2.577907;
   DATA[353,1] := 529.2057;
   DATA[353,2] := 2.0;
   DATA[353,3] := 2.0;
   DATA[353,4] := 262.0482;
   DATA[353,5] := 8.391951;
   DATA[353,6] := 328.3004;
   DATA[353,7] := 2.439496;
   DATA[353,8] := 2.0;
   DATA[353,9] := 2.0;
   DATA[353,10] := 2.0;
   DATA[353,11] := 19.65235;
   DATA[353,12] := 2.209525;
   DATA[353,13] := 972.2267;
   DATA[353,14] := 1.0;
   DATA[353,15] := 2.0;
   DATA[353,16] := 1.0;
   DATA[353,17] := 1.0;
   DATA[353,18] := 1.0;
   DATA[353,19] := 2.0;
   DATA[353,20] := 148.808;
   DATA[353,21] := 155.96;
   DATA[353,22] := 1.716464;
   DATA[353,23] := 969.9052;
   DATA[353,24] := 2.0;
   DATA[353,25] := 2.0;
   DATA[353,26] := 7.879582;
   DATA[353,27] := 145.0397;
   DATA[353,28] := 263.7465;
   DATA[353,29] := 12.15073;
   DATA[353,30] := 1.724045;
   DATA[353,31] := 1.277059;
   DATA[353,32] := 0.7347566;
   DATA[353,33] := 0.3086186;
   DATA[353,34] := 2.0;
   DATA[353,35] := 250.785;
   DATA[353,36] := 1.617916;
   DATA[353,37] := 189.4546;
   DATA[353,38] := 0.000128152;
   DATA[353,39] := 1.0;
   DATA[354,0] := 2.562534;
   DATA[354,1] := 528.9309;
   DATA[354,2] := 2.0;
   DATA[354,3] := 2.0;
   DATA[354,4] := 262.0482;
   DATA[354,5] := 8.391951;
   DATA[354,6] := 328.3004;
   DATA[354,7] := 2.439496;
   DATA[354,8] := 2.0;
   DATA[354,9] := 2.0;
   DATA[354,10] := 2.0;
   DATA[354,11] := 19.65235;
   DATA[354,12] := 2.209525;
